short summary
==================
This test method tests ``assert.integer.unsigned.x.valueIsOdd``
of CNM_AssertionInterfaces library, 
it provides the possibility to handover test data via parameter 


.. <legal notes>

legal notes
=================
| SPDX-FileCopyrightText: © 2022 ekvip automation GmbH <info@ekvip.de>
| SPDX-License-Identifier: Apache-2.0
| For details check: Apache-2.0_

.. _Apache-2.0: https://www.apache.org/licenses/LICENSE-2.0

.. </legal notes>

parameters
==========

*)

METHOD testValueIsOdd
VAR_INPUT
	(* for the test it's the parameter ``currentValue`` *)
	valueToTest	:__UXINT;
END_VAR
VAR
	(* just the expectation if the assertion to test must be worng or true *)
	assertionIsWrong		:BOOL;
	(* contains the format string for the test message *)
	message					:Tc2_System.T_MaxString;
	(* TwinCAT printf with the test message *)
	messageStringBuilder	:Tc2_Utilities.FB_FormatString;
END_VAR
THIS^.assertorContainer.resetAssertor();

assertionIsWrong := (NOT valueToTest.FIRST_BIT);

message := SEL(
	assertionIsWrong,
	'currentValue is %d assertion must be TRUE',
	'currentValue is %d assertion must be FALSE'
);

messageStringBuilder(
	sFormat := message,
	arg1 := THIS^.AnyToArg(valueToTest)
);

THIS^.assertorContainer.assertor.assert.integer.unsigned.x.valueIsOdd(
	currentValue 	:= valueToTest,
	message			:= ''  
); 

THIS^.AssertEquals_BOOL(
	Expected 	:= assertionIsWrong,
	Actual 		:= THIS^.assertorContainer.wasAssertionWrong,
	Message 	:= messageStringBuilder.sOut
);
END_METHOD

END_FUNCTION_BLOCK

// ---- AssertionTester/AssertionTests/IntegerAssertions/classes/XintAssertionTests.TcPOU
(*

short summary
==================
This class tests all methods of xint assertions
with various combinations of inputs and checks expected 
outputs are satisfied or not

.. <legal notes>

legal notes
=================
| SPDX-FileCopyrightText: © 2022 ekvip automation GmbH <info@ekvip.de>
| SPDX-License-Identifier: Apache-2.0
| For details check: Apache-2.0_

.. _Apache-2.0: https://www.apache.org/licenses/LICENSE-2.0

.. </legal notes>

methods and properties
======================

*)

FUNCTION_BLOCK XintAssertionTests EXTENDS AbstractAssertorTest
VAR_INPUT
END_VAR
VAR CONSTANT
	(* prefix to unify the test names *)
	TEST_NAME_PREFIX	:Tc2_System.T_MaxString := 'assert.integer.signed.x.';
	(* number of the lsb *)
	FIRST_BIT				:USINT := 0;
	(* number of the msb *)
	LAST_BIT				:USINT := ((SIZEOF(__XINT)*8)-1);
	(* since we don't know the lenght of __XINT we need it to initialize ``MULTIPLICAND`` *)
	{attribute 'hide'}
	INIT_VALUE_MULTIPLICAND	:__XWORD := 16#1111_1111;
	(* multiplicand for the ``multiplier`` *)
	{warning disable C0196}
	MULTIPLICAND			:__XINT := (ROR(INIT_VALUE_MULTIPLICAND, 32) OR INIT_VALUE_MULTIPLICAND);
	{warning enable C0196}
	(* first of all multipliers the test iterates *)
	FIRST_MULTIPLIER		:__XINT := 0;
	(* first of all multipliers the test iterates *)
	LAST_MULTIPLIER			:__XINT := 15;
	(* just the value zero *)
	ZERO					:__XINT := 0;
	(* just the lsb is set, it's just the value one *)
	LSB_ONLY				:__XINT := 1;
	(* all bits are set *)
	ALL_BITS_SET			:__XINT := -1;
	(* the msb is set only *)
	MINIMUM_VALUE			:__XINT := ROR(LSB_ONLY,1);
	(* 
	since we don't know the lenght of __XINT 
	we need it to initialize ``MAXIMUM_VALUE``.
	SHR is not working with __XINT
	*)
	{attribute 'hide'}
	{warning disable C0195}
	BINARY_MINUS_ONE		:__XWORD := ALL_BITS_SET;
	{warning enable C0195}
	(* the msb is unset only *)
	{warning disable C0196}
	MAXIMUM_VALUE			:__XINT := SHR(BINARY_MINUS_ONE,1);
	{warning ensable C0196}
END_VAR

THIS^.runValueIsEqualToTests();
THIS^.runValueIsEvenTests();
THIS^.runValueIsGreaterTests();
THIS^.runValueIsInRangeOfTests();
THIS^.runValueIsLessThanTests();
THIS^.runValueIsMaxTests();
THIS^.runValueIsMinTests();
THIS^.runValueIsNegativeTests();
THIS^.runValueIsNotEqualToTests();
THIS^.runValueIsOddTests();
THIS^.runValueIsPositiveTests();

(*

short summary
==================
This test method is a helper function to create a unified test name

.. <legal notes>

legal notes
=================
| SPDX-FileCopyrightText: © 2022 ekvip automation GmbH <info@ekvip.de>
| SPDX-License-Identifier: Apache-2.0
| For details check: Apache-2.0_

.. _Apache-2.0: https://www.apache.org/licenses/LICENSE-2.0

.. </legal notes>

parameters
==========

*)

METHOD PROTECTED getTestNameFor :Tc2_System.T_MaxString
VAR_INPUT
	(* name of the method to test, to create a unified test name *)
	nameOfMethodToTest	:Tc2_System.T_MaxString;
END_VAR
getTestNameFor := Tc2_Standard.CONCAT(THIS^.TEST_NAME_PREFIX, nameOfMethodToTest);
END_METHOD

(*

short summary
==================
This test method tests ``assert.integer.signed.x.valueIsEqualTo``
method of CNM_AssertionInterfaces library with various inputs

.. <legal notes>

legal notes
=================
| SPDX-FileCopyrightText: © 2022 ekvip automation GmbH <info@ekvip.de>
| SPDX-License-Identifier: Apache-2.0
| For details check: Apache-2.0_

.. _Apache-2.0: https://www.apache.org/licenses/LICENSE-2.0

.. </legal notes>

*)

METHOD runValueIsEqualToTests
RETURN (NOT TcUnit.TEST_ORDERED(THIS^.getTestNameFor('valueIsEqualTo')));

THIS^.testValueIsEqualTo(
	valueToTest := THIS^.ZERO,
	expected := THIS^.ALL_BITS_SET
);
THIS^.testValueIsEqualTo(
	valueToTest := THIS^.ZERO,
	expected := THIS^.ZERO
);
THIS^.testValueIsEqualTo(
	valueToTest := THIS^.ALL_BITS_SET,
	expected := THIS^.ALL_BITS_SET
);
THIS^.testValueIsEqualTo(
	valueToTest := THIS^.ALL_BITS_SET,
	expected := THIS^.ZERO
);
THIS^.testValueIsEqualTo(
	valueToTest := THIS^.LSB_ONLY,
	expected := THIS^.LSB_ONLY
);
THIS^.testValueIsEqualTo(
	valueToTest := THIS^.LSB_ONLY,
	expected := THIS^.MINIMUM_VALUE
);
THIS^.testValueIsEqualTo(
	valueToTest := THIS^.MINIMUM_VALUE,
	expected := THIS^.MINIMUM_VALUE
);
THIS^.testValueIsEqualTo(
	valueToTest := THIS^.MINIMUM_VALUE,
	expected := THIS^.LSB_ONLY
);
THIS^.testValueIsEqualTo(
	valueToTest := THIS^.MINIMUM_VALUE,
	expected := THIS^.MAXIMUM_VALUE
);

TcUnit.TEST_FINISHED();
END_METHOD

(*

short summary
==================
This test method tests ``assert.integer.signed.x.valueIsEven``
of CNM_AssertionInterfaces library with various inputs

.. <legal notes>

legal notes
=================
| SPDX-FileCopyrightText: © 2022 ekvip automation GmbH <info@ekvip.de>
| SPDX-License-Identifier: Apache-2.0
| For details check: Apache-2.0_

.. _Apache-2.0: https://www.apache.org/licenses/LICENSE-2.0

.. </legal notes>

*)

METHOD runValueIsEvenTests
VAR
	(* it's just part of the test data *)
	valueToTest	:__XINT;
	(* multiplier to get various bit patterns *)
	multiplier	:__XINT;
END_VAR
RETURN (NOT TcUnit.TEST_ORDERED(THIS^.getTestNameFor('valueIsEven')));

FOR multiplier := THIS^.FIRST_MULTIPLIER TO THIS^.LAST_MULTIPLIER DO
	valueToTest := (THIS^.MULTIPLICAND * multiplier);
	THIS^.testValueIsEven(
		valueToTest := valueToTest
	);
END_FOR

TcUnit.TEST_FINISHED();
END_METHOD

(*

short summary
==================
This test method tests ``assert.integer.signed.x.valueIsGreaterThan``
method of CNM_AssertionInterfaces library with various inputs

.. <legal notes>

legal notes
=================
| SPDX-FileCopyrightText: © 2022 ekvip automation GmbH <info@ekvip.de>
| SPDX-License-Identifier: Apache-2.0
| For details check: Apache-2.0_

.. _Apache-2.0: https://www.apache.org/licenses/LICENSE-2.0

.. </legal notes>

*)

METHOD runValueIsGreaterTests
RETURN (NOT TcUnit.TEST_ORDERED(THIS^.getTestNameFor('valueIsGreaterThan')));

THIS^.testValueIsGreater(
	valueToTest := THIS^.ZERO,
	less := THIS^.ALL_BITS_SET
);
THIS^.testValueIsGreater(
	valueToTest := THIS^.ZERO,
	less := THIS^.ZERO
);
THIS^.testValueIsGreater(
	valueToTest := THIS^.ALL_BITS_SET,
	less := THIS^.ALL_BITS_SET
);
THIS^.testValueIsGreater(
	valueToTest := THIS^.ALL_BITS_SET,
	less := THIS^.ZERO
);
THIS^.testValueIsGreater(
	valueToTest := THIS^.LSB_ONLY,
	less := THIS^.LSB_ONLY
);
THIS^.testValueIsGreater(
	valueToTest := THIS^.LSB_ONLY,
	less := THIS^.ZERO
);
THIS^.testValueIsGreater(
	valueToTest := THIS^.LSB_ONLY,
	less := (THIS^.LSB_ONLY+THIS^.LSB_ONLY)
);
THIS^.testValueIsGreater(
	valueToTest := THIS^.MINIMUM_VALUE,
	less := THIS^.MINIMUM_VALUE
);
THIS^.testValueIsGreater(
	valueToTest := THIS^.MINIMUM_VALUE,
	less := THIS^.ALL_BITS_SET
);
THIS^.testValueIsGreater(
	valueToTest := THIS^.MINIMUM_VALUE,
	less := THIS^.MAXIMUM_VALUE
);
THIS^.testValueIsGreater(
	valueToTest := THIS^.MAXIMUM_VALUE,
	less := THIS^.MINIMUM_VALUE
);

TcUnit.TEST_FINISHED();
END_METHOD

(*

short summary
==================
This test method tests ``assert.integer.signed.x.valueIsInRangeOf``
method of CNM_AssertionInterfaces library with various inputs

.. <legal notes>

legal notes
=================
| SPDX-FileCopyrightText: © 2022 ekvip automation GmbH <info@ekvip.de>
| SPDX-License-Identifier: Apache-2.0
| For details check: Apache-2.0_

.. _Apache-2.0: https://www.apache.org/licenses/LICENSE-2.0

.. </legal notes>

*)

METHOD runValueIsInRangeOfTests
RETURN (NOT TcUnit.TEST_ORDERED(THIS^.getTestNameFor('valueIsInRangeOf')));

THIS^.testValueIsInRangeOf(
	lower := THIS^.ZERO,
	valueToTest := THIS^.LSB_ONLY,
	upper := THIS^.ALL_BITS_SET
);
THIS^.testValueIsInRangeOf(
	lower := THIS^.ZERO,
	valueToTest := THIS^.ZERO,
	upper := THIS^.ZERO
);
THIS^.testValueIsInRangeOf(
	lower := THIS^.ALL_BITS_SET,
	valueToTest := THIS^.ALL_BITS_SET,
	upper := THIS^.ALL_BITS_SET
);
THIS^.testValueIsInRangeOf(
	lower := THIS^.ALL_BITS_SET,
	valueToTest := THIS^.LSB_ONLY,
	upper := THIS^.ZERO
);
THIS^.testValueIsInRangeOf(
	lower := THIS^.ALL_BITS_SET,
	valueToTest := THIS^.ZERO,
	upper := THIS^.ZERO
);
THIS^.testValueIsInRangeOf(
	lower := THIS^.MAXIMUM_VALUE,
	valueToTest := THIS^.ZERO,
	upper := THIS^.MINIMUM_VALUE
);
THIS^.testValueIsInRangeOf(
	lower := THIS^.MINIMUM_VALUE,
	valueToTest := THIS^.ZERO,
	upper := THIS^.MAXIMUM_VALUE
);
THIS^.testValueIsInRangeOf(
	lower := THIS^.MAXIMUM_VALUE,
	valueToTest := THIS^.MINIMUM_VALUE,
	upper := THIS^.MINIMUM_VALUE
);
THIS^.testValueIsInRangeOf(
	lower := THIS^.MINIMUM_VALUE,
	valueToTest := THIS^.MAXIMUM_VALUE,
	upper := THIS^.MAXIMUM_VALUE
);
THIS^.testValueIsInRangeOf(
	lower := THIS^.MINIMUM_VALUE,
	valueToTest := THIS^.MINIMUM_VALUE,
	upper := THIS^.MAXIMUM_VALUE
);

TEST_FINISHED();
END_METHOD

(*

short summary
==================
This test method tests ``assert.integer.signed.x.valueIsLessThan``
method of CNM_AssertionInterfaces library with various inputs

.. <legal notes>

legal notes
=================
| SPDX-FileCopyrightText: © 2022 ekvip automation GmbH <info@ekvip.de>
| SPDX-License-Identifier: Apache-2.0
| For details check: Apache-2.0_

.. _Apache-2.0: https://www.apache.org/licenses/LICENSE-2.0

.. </legal notes>

*)

METHOD runValueIsLessThanTests
RETURN (NOT TcUnit.TEST_ORDERED(THIS^.getTestNameFor('valueIsLessThan')));

THIS^.testValueIsLessThan(
	valueToTest := THIS^.ZERO,
	greater := THIS^.ALL_BITS_SET
);
THIS^.testValueIsLessThan(
	valueToTest := THIS^.ZERO,
	greater := THIS^.ZERO
);
THIS^.testValueIsLessThan(
	valueToTest := THIS^.ALL_BITS_SET,
	greater := THIS^.ALL_BITS_SET
);
THIS^.testValueIsLessThan(
	valueToTest := THIS^.ALL_BITS_SET,
	greater := THIS^.ZERO
);
THIS^.testValueIsLessThan(
	valueToTest := THIS^.LSB_ONLY,
	greater := THIS^.LSB_ONLY
);
THIS^.testValueIsLessThan(
	valueToTest := THIS^.LSB_ONLY,
	greater := THIS^.ZERO
);
THIS^.testValueIsLessThan(
	valueToTest := THIS^.MINIMUM_VALUE,
	greater := (THIS^.MINIMUM_VALUE+THIS^.LSB_ONLY)
);
THIS^.testValueIsLessThan(
	valueToTest := THIS^.MINIMUM_VALUE,
	greater := THIS^.MINIMUM_VALUE
);
THIS^.testValueIsLessThan(
	valueToTest := THIS^.MINIMUM_VALUE,
	greater := THIS^.ALL_BITS_SET
);
THIS^.testValueIsLessThan(
	valueToTest := THIS^.MINIMUM_VALUE,
	greater := THIS^.MAXIMUM_VALUE
);
THIS^.testValueIsLessThan(
	valueToTest := THIS^.MAXIMUM_VALUE,
	greater := THIS^.MINIMUM_VALUE
);

TcUnit.TEST_FINISHED();
END_METHOD

(*

short summary
==================
This test method tests ``assert.integer.signed.x.valueIsMax``
method of CNM_AssertionInterfaces library with various inputs

.. <legal notes>

legal notes
=================
| SPDX-FileCopyrightText: © 2022 ekvip automation GmbH <info@ekvip.de>
| SPDX-License-Identifier: Apache-2.0
| For details check: Apache-2.0_

.. _Apache-2.0: https://www.apache.org/licenses/LICENSE-2.0

.. </legal notes>

*)

METHOD runValueIsMaxTests
RETURN (NOT TcUnit.TEST_ORDERED(THIS^.getTestNameFor('valueIsMax')));

THIS^.testValueIsMax(
	valueToTest := THIS^.ZERO,
	maximum := THIS^.LSB_ONLY
);
THIS^.testValueIsMax(
	valueToTest := THIS^.LSB_ONLY,
	maximum := THIS^.ZERO
);
THIS^.testValueIsMax(
	valueToTest := THIS^.ZERO,
	maximum := THIS^.ZERO
);
THIS^.testValueIsMax(
	valueToTest := THIS^.ALL_BITS_SET,
	maximum := ALL_BITS_SET
);
THIS^.testValueIsMax(
	valueToTest := (THIS^.ALL_BITS_SET-THIS^.LSB_ONLY),
	maximum := THIS^.ALL_BITS_SET
);
THIS^.testValueIsMax(
	valueToTest := THIS^.ALL_BITS_SET,
	maximum := (THIS^.ALL_BITS_SET-THIS^.LSB_ONLY)
);
THIS^.testValueIsMax(
	valueToTest := THIS^.MINIMUM_VALUE,
	maximum := (THIS^.MINIMUM_VALUE+THIS^.LSB_ONLY)
);
THIS^.testValueIsMax(
	valueToTest := (THIS^.MINIMUM_VALUE+THIS^.LSB_ONLY),
	maximum := THIS^.MINIMUM_VALUE
);
THIS^.testValueIsMax(
	valueToTest := THIS^.MINIMUM_VALUE,
	maximum := THIS^.MINIMUM_VALUE
);
THIS^.testValueIsMax(
	valueToTest := THIS^.MINIMUM_VALUE,
	maximum := THIS^.MAXIMUM_VALUE
);
THIS^.testValueIsMax(
	valueToTest := THIS^.MAXIMUM_VALUE,
	maximum := THIS^.MINIMUM_VALUE
);

TcUnit.TEST_FINISHED();
END_METHOD

(*

short summary
==================
This test method tests ``assert.integer.signed.x.valueIsMin``
method of CNM_AssertionInterfaces library with various inputs

.. <legal notes>

legal notes
=================
| SPDX-FileCopyrightText: © 2022 ekvip automation GmbH <info@ekvip.de>
| SPDX-License-Identifier: Apache-2.0
| For details check: Apache-2.0_

.. _Apache-2.0: https://www.apache.org/licenses/LICENSE-2.0

.. </legal notes>

*)

METHOD runValueIsMinTests
RETURN (NOT TcUnit.TEST_ORDERED(THIS^.getTestNameFor('valueIsMin')));

THIS^.testValueIsMin(
	valueToTest := THIS^.ZERO,
	minimum := THIS^.LSB_ONLY
);
THIS^.testValueIsMin(
	valueToTest := THIS^.LSB_ONLY,
	minimum := THIS^.ZERO
);
THIS^.testValueIsMin(
	valueToTest := THIS^.ZERO,
	minimum := THIS^.ZERO
);
THIS^.testValueIsMin(
	valueToTest := THIS^.ALL_BITS_SET,
	minimum := ALL_BITS_SET
);
THIS^.testValueIsMin(
	valueToTest := (THIS^.ALL_BITS_SET-THIS^.LSB_ONLY),
	minimum := THIS^.ALL_BITS_SET
);
THIS^.testValueIsMin(
	valueToTest := THIS^.ALL_BITS_SET,
	minimum := (THIS^.ALL_BITS_SET-THIS^.LSB_ONLY)
);
THIS^.testValueIsMin(
	valueToTest := THIS^.MINIMUM_VALUE,
	minimum := (THIS^.MINIMUM_VALUE+THIS^.LSB_ONLY)
);
THIS^.testValueIsMin(
	valueToTest := (THIS^.MINIMUM_VALUE+THIS^.LSB_ONLY),
	minimum := THIS^.MINIMUM_VALUE
);
THIS^.testValueIsMin(
	valueToTest := THIS^.MINIMUM_VALUE,
	minimum := THIS^.MINIMUM_VALUE
);
THIS^.testValueIsMin(
	valueToTest := THIS^.MINIMUM_VALUE,
	minimum := THIS^.MAXIMUM_VALUE
);
THIS^.testValueIsMin(
	valueToTest := THIS^.MAXIMUM_VALUE,
	minimum := THIS^.MINIMUM_VALUE
);

TcUnit.TEST_FINISHED();
END_METHOD

(*

short summary
==================
This test method tests ``assert.integer.signed.x.valueIsNegative``
of CNM_AssertionInterfaces library with various inputs

.. <legal notes>

legal notes
=================
| SPDX-FileCopyrightText: © 2022 ekvip automation GmbH <info@ekvip.de>
| SPDX-License-Identifier: Apache-2.0
| For details check: Apache-2.0_

.. _Apache-2.0: https://www.apache.org/licenses/LICENSE-2.0

.. </legal notes>

*)

METHOD runValueIsNegativeTests
VAR
	(* it's just part of the test data *)
	valueToTest	:__XINT;
	(* multiplier to get various bit patterns *)
	multiplier	:__XINT;
END_VAR
RETURN (NOT TcUnit.TEST_ORDERED(THIS^.getTestNameFor('valueIsNegative')));

FOR multiplier := THIS^.FIRST_MULTIPLIER TO THIS^.LAST_MULTIPLIER DO
	valueToTest := (THIS^.MULTIPLICAND * multiplier);
	THIS^.testValueIsNegative(
		valueToTest := valueToTest
	);
END_FOR

TcUnit.TEST_FINISHED();
END_METHOD

(*

short summary
==================
This test method tests ``assert.integer.signed.x.valueIsNotEqualTo``
method of CNM_AssertionInterfaces library with various inputs

.. <legal notes>

legal notes
=================
| SPDX-FileCopyrightText: © 2022 ekvip automation GmbH <info@ekvip.de>
| SPDX-License-Identifier: Apache-2.0
| For details check: Apache-2.0_

.. _Apache-2.0: https://www.apache.org/licenses/LICENSE-2.0

.. </legal notes>

*)

METHOD runValueIsNotEqualToTests
RETURN (NOT TcUnit.TEST_ORDERED(THIS^.getTestNameFor('valueIsNotEqualTo')));

THIS^.testValueIsNotEqualTo(
	valueToTest := THIS^.ZERO,
	unexpected := THIS^.ALL_BITS_SET
);
THIS^.testValueIsNotEqualTo(
	valueToTest := THIS^.ZERO,
	unexpected := THIS^.ZERO
);
THIS^.testValueIsNotEqualTo(
	valueToTest := THIS^.ALL_BITS_SET,
	unexpected := THIS^.ALL_BITS_SET
);
THIS^.testValueIsNotEqualTo(
	valueToTest := THIS^.ALL_BITS_SET,
	unexpected := THIS^.ZERO
);
THIS^.testValueIsNotEqualTo(
	valueToTest := THIS^.LSB_ONLY,
	unexpected := THIS^.LSB_ONLY
);
THIS^.testValueIsNotEqualTo(
	valueToTest := THIS^.LSB_ONLY,
	unexpected := THIS^.MINIMUM_VALUE
);
THIS^.testValueIsNotEqualTo(
	valueToTest := THIS^.MINIMUM_VALUE,
	unexpected := THIS^.MINIMUM_VALUE
);
THIS^.testValueIsNotEqualTo(
	valueToTest := THIS^.MINIMUM_VALUE,
	unexpected := THIS^.LSB_ONLY
);
THIS^.testValueIsNotEqualTo(
	valueToTest := THIS^.MINIMUM_VALUE,
	unexpected := THIS^.MAXIMUM_VALUE
);

TcUnit.TEST_FINISHED();
END_METHOD

(*

short summary
==================
This test method tests ``assert.integer.signed.x.valueIsOdd``
of CNM_AssertionInterfaces library with various inputs

.. <legal notes>

legal notes
=================
| SPDX-FileCopyrightText: © 2022 ekvip automation GmbH <info@ekvip.de>
| SPDX-License-Identifier: Apache-2.0
| For details check: Apache-2.0_

.. _Apache-2.0: https://www.apache.org/licenses/LICENSE-2.0

.. </legal notes>

*)

METHOD runValueIsOddTests
VAR
	(* it's just part of the test data *)
	valueToTest	:__XINT;
	(* multiplier to get various bit patterns *)
	multiplier	:__XINT;
END_VAR
RETURN (NOT TcUnit.TEST_ORDERED(THIS^.getTestNameFor('valueIsOdd')));

FOR multiplier := THIS^.FIRST_MULTIPLIER TO THIS^.LAST_MULTIPLIER DO
	valueToTest := (THIS^.MULTIPLICAND * multiplier);
	THIS^.testValueIsOdd(
		valueToTest := valueToTest
	);
END_FOR

TcUnit.TEST_FINISHED();
END_METHOD

(*

short summary
==================
This test method tests ``assert.integer.signed.x.valueIsPositive``
of CNM_AssertionInterfaces library with various inputs

.. <legal notes>

legal notes
=================
| SPDX-FileCopyrightText: © 2022 ekvip automation GmbH <info@ekvip.de>
| SPDX-License-Identifier: Apache-2.0
| For details check: Apache-2.0_

.. _Apache-2.0: https://www.apache.org/licenses/LICENSE-2.0

.. </legal notes>

*)

METHOD runValueIsPositiveTests
VAR
	(* it's just part of the test data *)
	valueToTest	:__XINT;
	(* multiplier to get various bit patterns *)
	multiplier	:__XINT;
END_VAR
RETURN (NOT TcUnit.TEST_ORDERED(THIS^.getTestNameFor('valueIsPositive')));

FOR multiplier := THIS^.FIRST_MULTIPLIER TO THIS^.LAST_MULTIPLIER DO
	valueToTest := (THIS^.MULTIPLICAND * multiplier);
	THIS^.testValueIsPositive(
		valueToTest := valueToTest
	);
END_FOR

TcUnit.TEST_FINISHED();
END_METHOD

(*

short summary
==================
This test method tests ``assert.integer.signed.x.valueIsEqualTo``
method of CNM_AssertionInterfaces library, 
it provides the possibility to handover test data via parameter 


.. <legal notes>

legal notes
=================
| SPDX-FileCopyrightText: © 2022 ekvip automation GmbH <info@ekvip.de>
| SPDX-License-Identifier: Apache-2.0
| For details check: Apache-2.0_

.. _Apache-2.0: https://www.apache.org/licenses/LICENSE-2.0

.. </legal notes>

parameters
==========

*)

METHOD testValueIsEqualTo
VAR_INPUT
	(* for the test it's the parameter ``currentValue`` *)
	valueToTest	:__XINT;
	(* for the test it's the parameter ``expectedValue`` *)
	expected	:__XINT;
END_VAR
VAR
	(* just the expectation if the assertion to test must be worng or true *)
	assertionIsWrong		:BOOL;
	(* contains the format string for the test message *)
	message					:Tc2_System.T_MaxString;
	(* TwinCAT printf with the test message *)
	messageStringBuilder	:Tc2_Utilities.FB_FormatString;
END_VAR
THIS^.assertorContainer.resetAssertor();

assertionIsWrong := (valueToTest <> expected);
message := SEL(
	assertionIsWrong,
	'currentValue is %d expectedValue is %d assertion must be TRUE', 
	'currentValue is %d expectedValue is %d assertion must be FALSE'
);
messageStringBuilder(
	sFormat := message,
	arg1 := THIS^.AnyToArg(valueToTest),
	arg2 := THIS^.AnyToArg(expected)
);

THIS^.assertorContainer.assertor.assert.integer.signed.x.valueIsEqualTo(
	currentValue := valueToTest,
	expectedValue := expected,
	message := ''
);

THIS^.AssertEquals_BOOL(
	Expected 	:= assertionIsWrong,
	Actual 		:= THIS^.assertorContainer.wasAssertionWrong,
	Message 	:= messageStringBuilder.sOut
);
END_METHOD

(*

short summary
==================
This test method tests ``assert.integer.signed.x.valueIsEven``
of CNM_AssertionInterfaces library, 
it provides the possibility to handover test data via parameter 


.. <legal notes>

legal notes
=================
| SPDX-FileCopyrightText: © 2022 ekvip automation GmbH <info@ekvip.de>
| SPDX-License-Identifier: Apache-2.0
| For details check: Apache-2.0_

.. _Apache-2.0: https://www.apache.org/licenses/LICENSE-2.0

.. </legal notes>

parameters
==========

*)

METHOD testValueIsEven
VAR_INPUT
	(* for the test it's the parameter ``currentValue`` *)
	valueToTest	:__XINT;
END_VAR
VAR
	(* just the expectation if the assertion to test must be worng or true *)
	assertionIsWrong		:BOOL;
	(* contains the format string for the test message *)
	message					:Tc2_System.T_MaxString;
	(* TwinCAT printf with the test message *)
	messageStringBuilder	:Tc2_Utilities.FB_FormatString;
END_VAR
THIS^.assertorContainer.resetAssertor();

assertionIsWrong := (valueToTest.FIRST_BIT);

message := SEL(
	assertionIsWrong,
	'currentValue is %d assertion must be TRUE',
	'currentValue is %d assertion must be FALSE'
);

messageStringBuilder(
	sFormat := message,
	arg1 := THIS^.AnyToArg(valueToTest)
);

THIS^.assertorContainer.assertor.assert.integer.signed.x.valueIsEven(
	currentValue 	:= valueToTest,
	message			:= ''  
); 

THIS^.AssertEquals_BOOL(
	Expected 	:= assertionIsWrong,
	Actual 		:= THIS^.assertorContainer.wasAssertionWrong,
	Message 	:= messageStringBuilder.sOut
);
END_METHOD

(*

short summary
==================
This test method tests ``assert.integer.signed.x.valueIsGreaterThan``
method of CNM_AssertionInterfaces library, 
it provides the possibility to handover test data via parameter 


.. <legal notes>

legal notes
=================
| SPDX-FileCopyrightText: © 2022 ekvip automation GmbH <info@ekvip.de>
| SPDX-License-Identifier: Apache-2.0
| For details check: Apache-2.0_

.. _Apache-2.0: https://www.apache.org/licenses/LICENSE-2.0

.. </legal notes>

parameters
==========

*)

METHOD testValueIsGreater
VAR_INPUT
	(* for the test it's the parameter ``currentValue`` *)
	valueToTest	:__XINT;
	(* for the test it's the parameter ``lessValue`` *)
	less		:__XINT;
END_VAR
VAR
	(* just the expectation if the assertion to test must be worng or true *)
	assertionIsWrong		:BOOL;
	(* contains the format string for the test message *)
	message					:Tc2_System.T_MaxString;
	(* TwinCAT printf with the test message *)
	messageStringBuilder	:Tc2_Utilities.FB_FormatString;
END_VAR
THIS^.assertorContainer.resetAssertor();

assertionIsWrong := (valueToTest <= less);
message := SEL(
	assertionIsWrong,
	'currentValue is %d lessValue is %d assertion must be TRUE', 
	'currentValue is %d lessValue is %d assertion must be FALSE'
);
messageStringBuilder(
	sFormat := message,
	arg1 := THIS^.AnyToArg(valueToTest),
	arg2 := THIS^.AnyToArg(less)
);

THIS^.assertorContainer.assertor.assert.integer.signed.x.valueIsGreaterThan(
	currentValue := valueToTest,
	lessValue := less,
	message := ''
);

THIS^.AssertEquals_BOOL(
	Expected 	:= assertionIsWrong,
	Actual 		:= THIS^.assertorContainer.wasAssertionWrong,
	Message 	:= messageStringBuilder.sOut
);
END_METHOD

(*

short summary
==================
This test method tests ``assert.integer.signed.x.valueIsInRangeOf``
method of CNM_AssertionInterfaces library, 
it provides the possibility to handover test data via parameter 


.. <legal notes>

legal notes
=================
| SPDX-FileCopyrightText: © 2022 ekvip automation GmbH <info@ekvip.de>
| SPDX-License-Identifier: Apache-2.0
| For details check: Apache-2.0_

.. _Apache-2.0: https://www.apache.org/licenses/LICENSE-2.0

.. </legal notes>

parameters
==========

*)

METHOD testValueIsInRangeOf
VAR_INPUT
	(* for the test it's the parameter ``lowerLimit`` *)
	lower		:__XINT;
	(* for the test it's the parameter ``currentValue`` *)
	valueToTest	:__XINT;
	(* for the test it's the parameter ``upperLimit`` *)
	upper		:__XINT;
END_VAR          
VAR
	(* just the expectation if the assertion to test must be worng or true *)
	assertionIsWrong		:BOOL;
	(* contains the format string for the test message *)
	message					:Tc2_System.T_MaxString;
	(* TwinCAT printf with the test message *)
	messageStringBuilder	:Tc2_Utilities.FB_FormatString;
END_VAR
THIS^.assertorContainer.resetAssertor();

assertionIsWrong := ((valueToTest < lower) OR (valueToTest > upper)); 

message := SEL(
	assertionIsWrong,
	'lowerLimit is %d currentValue is %d upperLimit is %d assertion must be TRUE', 
	'lowerLimit is %d currentValue is %d upperLimit is %d assertion must be FALSE'
);

messageStringBuilder(
	sFormat := message,
	arg1 := THIS^.AnyToArg(lower),
	arg2 := THIS^.AnyToArg(valueToTest),
	arg3 := THIS^.AnyToArg(upper)
);

THIS^.assertorContainer.assertor.assert.integer.signed.x.valueIsInRangeOf(
	lowerLimit := lower,
	currentValue := valueToTest,
	upperLimit := upper,
	message := ''
);

THIS^.AssertEquals_BOOL(
	Expected 	:= assertionIsWrong,
	Actual 		:= THIS^.assertorContainer.wasAssertionWrong,
	Message 	:= messageStringBuilder.sOut
);
END_METHOD

(*

short summary
==================
This test method tests ``assert.integer.signed.x.valueIsLessThan``
method of CNM_AssertionInterfaces library, 
it provides the possibility to handover test data via parameter 


.. <legal notes>

legal notes
=================
| SPDX-FileCopyrightText: © 2022 ekvip automation GmbH <info@ekvip.de>
| SPDX-License-Identifier: Apache-2.0
| For details check: Apache-2.0_

.. _Apache-2.0: https://www.apache.org/licenses/LICENSE-2.0

.. </legal notes>

parameters
==========

*)

METHOD testValueIsLessThan
VAR_INPUT
	(* for the test it's the parameter ``currentValue`` *)
	valueToTest	:__XINT;
	(* for the test it's the parameter ``greaterValue`` *)
	greater		:__XINT;
END_VAR
VAR
	(* just the expectation if the assertion to test must be worng or true *)
	assertionIsWrong		:BOOL;
	(* contains the format string for the test message *)
	message					:Tc2_System.T_MaxString;
	(* TwinCAT printf with the test message *)
	messageStringBuilder	:Tc2_Utilities.FB_FormatString;
END_VAR
THIS^.assertorContainer.resetAssertor();

assertionIsWrong := (valueToTest >= greater);
message := SEL(
	assertionIsWrong,
	'currentValue is %d greaterValue is %d assertion must be TRUE',
	'currentValue is %d greaterValue is %d assertion must be FALSE'
);
messageStringBuilder(
	sFormat := message,
	arg1 := THIS^.AnyToArg(valueToTest),
	arg2 := THIS^.AnyToArg(greater)
);

THIS^.assertorContainer.assertor.assert.integer.signed.x.valueIsLessThan(
	currentValue := valueToTest,
	greaterValue := greater,
	message := ''
);

THIS^.AssertEquals_BOOL(
	Expected 	:= assertionIsWrong,
	Actual 		:= THIS^.assertorContainer.wasAssertionWrong,
	Message 	:= messageStringBuilder.sOut
);
END_METHOD

(*

short summary
==================
This test method tests ``assert.integer.signed.x.valueIsMax``
method of CNM_AssertionInterfaces library, 
it provides the possibility to handover test data via parameter 


.. <legal notes>

legal notes
=================
| SPDX-FileCopyrightText: © 2022 ekvip automation GmbH <info@ekvip.de>
| SPDX-License-Identifier: Apache-2.0
| For details check: Apache-2.0_

.. _Apache-2.0: https://www.apache.org/licenses/LICENSE-2.0

.. </legal notes>

parameters
==========

*)

METHOD testValueIsMax 
VAR_INPUT
	(* for the test it's the parameter ``currentValue`` *)
	valueToTest	:__XINT;
	(* for the test it's the parameter ``maximumValue`` *)
	maximum		:__XINT;
END_VAR
VAR
	(* just the expectation if the assertion to test must be worng or true *)
	assertionIsWrong		:BOOL;
	(* contains the format string for the test message *)
	message					:Tc2_System.T_MaxString;
	(* TwinCAT printf with the test message *)
	messageStringBuilder	:Tc2_Utilities.FB_FormatString;
END_VAR
THIS^.assertorContainer.resetAssertor();

assertionIsWrong := (valueToTest > maximum);
message := SEL(
	assertionIsWrong,
	'currentValue is %d maximumValue is %d assertion must be TRUE',
	'currentValue is %d maximumValue is %d assertion must be FALSE'
);
messageStringBuilder(
	sFormat := message,
	arg1 := THIS^.AnyToArg(valueToTest),
	arg2 := THIS^.AnyToArg(maximum)
);

THIS^.assertorContainer.assertor.assert.integer.signed.x.valueIsMax(
	currentValue := valueToTest,
	maximumValue := maximum,
	message := ''
);

THIS^.AssertEquals_BOOL(
	Expected 	:= assertionIsWrong,
	Actual 		:= THIS^.assertorContainer.wasAssertionWrong,
	Message 	:= messageStringBuilder.sOut
);
END_METHOD

(*

short summary
==================
This test method tests ``assert.integer.signed.x.valueIsMin``
method of CNM_AssertionInterfaces library, 
it provides the possibility to handover test data via parameter 


.. <legal notes>

legal notes
=================
| SPDX-FileCopyrightText: © 2022 ekvip automation GmbH <info@ekvip.de>
| SPDX-License-Identifier: Apache-2.0
| For details check: Apache-2.0_

.. _Apache-2.0: https://www.apache.org/licenses/LICENSE-2.0

.. </legal notes>

parameters
==========

*)

METHOD testValueIsMin 
VAR_INPUT
	(* for the test it's the parameter ``currentValue`` *)
	valueToTest	:__XINT;
	(* for the test it's the parameter ``minimumValue`` *)
	minimum		:__XINT;
END_VAR
VAR
	(* just the expectation if the assertion to test must be worng or true *)
	assertionIsWrong		:BOOL;
	(* contains the format string for the test message *)
	message					:Tc2_System.T_MaxString;
	(* TwinCAT printf with the test message *)
	messageStringBuilder	:Tc2_Utilities.FB_FormatString;
END_VAR
THIS^.assertorContainer.resetAssertor();

assertionIsWrong := (valueToTest < minimum);
message := SEL(
	assertionIsWrong,
	'currentValue is %d minimumValue is %d assertion must be TRUE',
	'currentValue is %d minimumValue is %d assertion must be FALSE'
);
messageStringBuilder(
	sFormat := message,
	arg1 := THIS^.AnyToArg(valueToTest),
	arg2 := THIS^.AnyToArg(minimum)
);

THIS^.assertorContainer.assertor.assert.integer.signed.x.valueIsMin(
	currentValue := valueToTest,
	minimumValue := minimum,
	message := ''
);

THIS^.AssertEquals_BOOL(
	Expected 	:= assertionIsWrong,
	Actual 		:= THIS^.assertorContainer.wasAssertionWrong,
	Message 	:= messageStringBuilder.sOut
);
END_METHOD

(*

short summary
==================
This test method tests ``assert.integer.signed.x.valueIsNegative``
of CNM_AssertionInterfaces library, 
it provides the possibility to handover test data via parameter 


.. <legal notes>

legal notes
=================
| SPDX-FileCopyrightText: © 2022 ekvip automation GmbH <info@ekvip.de>
| SPDX-License-Identifier: Apache-2.0
| For details check: Apache-2.0_

.. _Apache-2.0: https://www.apache.org/licenses/LICENSE-2.0

.. </legal notes>

parameters
==========

*)

METHOD testValueIsNegative
VAR_INPUT
	(* for the test it's the parameter ``currentValue`` *)
	valueToTest	:__XINT;
END_VAR
VAR
	(* just the expectation if the assertion to test must be worng or true *)
	assertionIsWrong		:BOOL;
	(* contains the format string for the test message *)
	message					:Tc2_System.T_MaxString;
	(* TwinCAT printf with the test message *)
	messageStringBuilder	:Tc2_Utilities.FB_FormatString;
END_VAR
THIS^.assertorContainer.resetAssertor();

assertionIsWrong := (valueToTest >= THIS^.ZERO);

message := SEL(
	assertionIsWrong,
	'currentValue is %d assertion must be TRUE',
	'currentValue is %d assertion must be FALSE'
);

messageStringBuilder(
	sFormat := message,
	arg1 := THIS^.AnyToArg(valueToTest)
);

THIS^.assertorContainer.assertor.assert.integer.signed.x.valueIsNegative(
	currentValue 	:= valueToTest,
	message			:= ''  
); 

THIS^.AssertEquals_BOOL(
	Expected 	:= assertionIsWrong,
	Actual 		:= THIS^.assertorContainer.wasAssertionWrong,
	Message 	:= messageStringBuilder.sOut
);
END_METHOD

(*

short summary
==================
This test method tests ``assert.integer.signed.x.valueIsNotEqualTo``
method of CNM_AssertionInterfaces library, 
it provides the possibility to handover test data via parameter 


.. <legal notes>

legal notes
=================
| SPDX-FileCopyrightText: © 2022 ekvip automation GmbH <info@ekvip.de>
| SPDX-License-Identifier: Apache-2.0
| For details check: Apache-2.0_

.. _Apache-2.0: https://www.apache.org/licenses/LICENSE-2.0

.. </legal notes>

parameters
==========

*)

METHOD testValueIsNotEqualTo
VAR_INPUT
	(* for the test it's the parameter ``currentValue`` *)
	valueToTest	:__XINT;
	(* for the test it's the parameter ``unexpectedValue`` *)
	unexpected	:__XINT;
END_VAR
VAR
	(* just the expectation if the assertion to test must be worng or true *)
	assertionIsWrong		:BOOL;
	(* contains the format string for the test message *)
	message					:Tc2_System.T_MaxString;
	(* TwinCAT printf with the test message *)
	messageStringBuilder	:Tc2_Utilities.FB_FormatString;
END_VAR
THIS^.assertorContainer.resetAssertor();

assertionIsWrong := (valueToTest = unexpected);
message := SEL(
	assertionIsWrong,
	'currentValue is %d unexpectedValue is %d assertion must be TRUE', 
	'currentValue is %d unexpectedValue is %d assertion must be FALSE'
);
messageStringBuilder(
	sFormat := message,
	arg1 := THIS^.AnyToArg(valueToTest),
	arg2 := THIS^.AnyToArg(unexpected)
);

THIS^.assertorContainer.assertor.assert.integer.signed.x.valueIsNotEqualTo(
	currentValue := valueToTest,
	unexpectedValue := unexpected,
	message := ''
);

THIS^.AssertEquals_BOOL(
	Expected 	:= assertionIsWrong,
	Actual 		:= THIS^.assertorContainer.wasAssertionWrong,
	Message 	:= messageStringBuilder.sOut
);
END_METHOD

(*

short summary
==================
This test method tests ``assert.integer.signed.x.valueIsOdd``
of CNM_AssertionInterfaces library, 
it provides the possibility to handover test data via parameter 


.. <legal notes>

legal notes
=================
| SPDX-FileCopyrightText: © 2022 ekvip automation GmbH <info@ekvip.de>
| SPDX-License-Identifier: Apache-2.0
| For details check: Apache-2.0_

.. _Apache-2.0: https://www.apache.org/licenses/LICENSE-2.0

.. </legal notes>

parameters
==========

*)

METHOD testValueIsOdd
VAR_INPUT
	(* for the test it's the parameter ``currentValue`` *)
	valueToTest	:__XINT;
END_VAR
VAR
	(* just the expectation if the assertion to test must be worng or true *)
	assertionIsWrong		:BOOL;
	(* contains the format string for the test message *)
	message					:Tc2_System.T_MaxString;
	(* TwinCAT printf with the test message *)
	messageStringBuilder	:Tc2_Utilities.FB_FormatString;
END_VAR
THIS^.assertorContainer.resetAssertor();

assertionIsWrong := (NOT valueToTest.FIRST_BIT);

message := SEL(
	assertionIsWrong,
	'currentValue is %d assertion must be TRUE',
	'currentValue is %d assertion must be FALSE'
);

messageStringBuilder(
	sFormat := message,
	arg1 := THIS^.AnyToArg(valueToTest)
);

THIS^.assertorContainer.assertor.assert.integer.signed.x.valueIsOdd(
	currentValue 	:= valueToTest,
	message			:= ''  
); 

THIS^.AssertEquals_BOOL(
	Expected 	:= assertionIsWrong,
	Actual 		:= THIS^.assertorContainer.wasAssertionWrong,
	Message 	:= messageStringBuilder.sOut
);
END_METHOD

(*

short summary
==================
This test method tests ``assert.integer.signed.x.valueIsPositive``
of CNM_AssertionInterfaces library, 
it provides the possibility to handover test data via parameter 


.. <legal notes>

legal notes
=================
| SPDX-FileCopyrightText: © 2022 ekvip automation GmbH <info@ekvip.de>
| SPDX-License-Identifier: Apache-2.0
| For details check: Apache-2.0_

.. _Apache-2.0: https://www.apache.org/licenses/LICENSE-2.0

.. </legal notes>

parameters
==========

*)

METHOD testValueIsPositive
VAR_INPUT
	(* for the test it's the parameter ``currentValue`` *)
	valueToTest	:__XINT;
END_VAR
VAR
	(* just the expectation if the assertion to test must be worng or true *)
	assertionIsWrong		:BOOL;
	(* contains the format string for the test message *)
	message					:Tc2_System.T_MaxString;
	(* TwinCAT printf with the test message *)
	messageStringBuilder	:Tc2_Utilities.FB_FormatString;
END_VAR
THIS^.assertorContainer.resetAssertor();

assertionIsWrong := (valueToTest < THIS^.ZERO);

message := SEL(
	assertionIsWrong,
	'currentValue is %d assertion must be TRUE',
	'currentValue is %d assertion must be FALSE'
);

messageStringBuilder(
	sFormat := message,
	arg1 := THIS^.AnyToArg(valueToTest)
);

THIS^.assertorContainer.assertor.assert.integer.signed.x.valueIsPositive(
	currentValue 	:= valueToTest,
	message			:= ''  
); 

THIS^.AssertEquals_BOOL(
	Expected 	:= assertionIsWrong,
	Actual 		:= THIS^.assertorContainer.wasAssertionWrong,
	Message 	:= messageStringBuilder.sOut
);
END_METHOD

END_FUNCTION_BLOCK

// ---- AssertionTester/AssertionTests/ObjectAssertions/classes/internal/ConcreteObject.TcPOU
(*

short summary
==================
Wraper Class for Object to make ´´isObjectValid()´´ calls possible
needed because ´´AbstractAssertorTest´´ already extends ´´FB_TestSuite´´

.. <legal notes>

legal notes
=================
| SPDX-FileCopyrightText: © 2022 ekvip automation GmbH <info@ekvip.de>
| SPDX-License-Identifier: Apache-2.0
| For details check: Apache-2.0_

.. _Apache-2.0: https://www.apache.org/licenses/LICENSE-2.0

.. </legal notes>

*)
FUNCTION_BLOCK ConcreteObject EXTENDS CNM_AbstractObject.Object
VAR
END_VAR

(*

short summary
=================
This abstract property returns the class name of the concrete object, 
which is useful to check the class name for ``__DELETE``.

.. <legal notes>

legal notes
=================
| SPDX-FileCopyrightText: © 2022 ekvip automation GmbH <info@ekvip.de>
| SPDX-License-Identifier: Apache-2.0
| For details check: Apache-2.0_

.. _Apache-2.0: https://www.apache.org/licenses/LICENSE-2.0

.. </legal notes>

*)


PROPERTY className : CNM_AbstractObject.ClassName
GET
className := 'ConcreteObject_Internal';
END_GET
END_PROPERTY

END_FUNCTION_BLOCK

// ---- AssertionTester/AssertionTests/ObjectAssertions/classes/internal/DWordValue.TcPOU
(*

short summary
==================
Implementaion of CNM_AbstractObject.IObject for testing purposes

.. <legal notes>

legal notes
=================
| SPDX-FileCopyrightText: © 2022 ekvip automation GmbH <info@ekvip.de>
| SPDX-License-Identifier: Apache-2.0
| For details check: Apache-2.0_

.. _Apache-2.0: https://www.apache.org/licenses/LICENSE-2.0

.. </legal notes>

*)

FUNCTION_BLOCK DWordValue EXTENDS CNM_AbstractObject.Object IMPLEMENTS IDWord

VAR
	(* local DWORD value of this Class*)
	dwordValue :DWORD;
END_VAR

(*

short summary
=================
This abstract property returns the class name of the concrete object, 
which is useful to check the class name for ``__DELETE``.

.. <legal notes>

legal notes
=================
| SPDX-FileCopyrightText: © 2022 ekvip automation GmbH <info@ekvip.de>
| SPDX-License-Identifier: Apache-2.0
| For details check: Apache-2.0_

.. _Apache-2.0: https://www.apache.org/licenses/LICENSE-2.0

.. </legal notes>

*)


PROPERTY className : CNM_AbstractObject.ClassName
GET
className := 'DWordValue_Internal';
END_GET
END_PROPERTY

(*

short summary
=================
overwrites compareTo of IObject: This method compares a foreign object with the own one, this is needed for sort orders.

.. <legal notes>

legal notes
=================
| SPDX-FileCopyrightText: © 2022 ekvip automation GmbH <info@ekvip.de>
| SPDX-License-Identifier: Apache-2.0
| For details check: Apache-2.0_

.. _Apache-2.0: https://www.apache.org/licenses/LICENSE-2.0

.. </legal notes>

parameters
=================
:return:``SMALLER``: ``THIS`` precedes in order,
``EQUAL``: ``THIS`` and ``object`` at the same position in order,
``GREATER``: ``THIS`` is after in order.
Checkout the library CNM_ReturnTypes.

*)

METHOD compareTo :CNM_ReturnTypes.ComparationResult
VAR_INPUT
	(* foreign objet to compare*)
	object		:CNM_AbstractObject.IObject;
END_VAR
VAR
	dwordObject	:IDWord;
END_VAR
IF (__QUERYINTERFACE(object, dwordObject)) THEN
	IF (THIS^.value < dwordObject.value) THEN
		compareTo := CNM_ReturnTypes.ComparationResult.SMALLER;
	ELSIF (THIS^.value = dwordObject.value) THEN
		compareTo := CNM_ReturnTypes.ComparationResult.EQUAL;
	ELSE
		compareTo := CNM_ReturnTypes.ComparationResult.GREATER;
	END_IF
ELSE
	compareTo := CNM_ReturnTypes.ComparationResult.SMALLER;
END_IF
END_METHOD

(*

short summary
=================
For initializing an DWordValue

.. <legal notes>

legal notes
=================
| SPDX-FileCopyrightText: © 2022 ekvip automation GmbH <info@ekvip.de>
| SPDX-License-Identifier: Apache-2.0
| For details check: Apache-2.0_

.. _Apache-2.0: https://www.apache.org/licenses/LICENSE-2.0

.. </legal notes>

parameters
=================

*)


METHOD FB_Init: BOOL
VAR_INPUT
	(* if TRUE, the retain variables are initialized (warm start / cold start) *)
    bInitRetains	:BOOL;
	(* if TRUE, the instance afterwards gets moved into the copy code (online change) *)
    bInCopyCode		:BOOL;
	(* value of the DWordValue Class*)
	initvalue 		:DWORD;
END_VAR
THIS^.dwordValue := initvalue;
END_METHOD

(*

short summary
=============
contains the DWORD Value of this Class

.. <legal notes>

legal notes
=================
| SPDX-FileCopyrightText: © 2023 ekvip automation GmbH <info@ekvip.de>
| SPDX-License-Identifier: Apache-2.0
| For details check: Apache-2.0_

.. _Apache-2.0: https://www.apache.org/licenses/LICENSE-2.0

.. </legal notes>

*)

PROPERTY value : DWORD
GET
value := THIS^.dwordValue;
END_GET
SET
THIS^.value := dwordValue;
END_SET
END_PROPERTY

END_FUNCTION_BLOCK

// ---- AssertionTester/AssertionTests/ObjectAssertions/classes/internal/ReverseOrderComparator.TcPOU
(*

short summary
=================
A comparator to reverse the natural order of the objects

.. <legal notes>

legal notes
=================
| SPDX-FileCopyrightText: © 2024 ekvip automation GmbH <info@ekvip.de>
| SPDX-License-Identifier: Apache-2.0
| For details check: Apache-2.0_

.. _Apache-2.0: https://www.apache.org/licenses/LICENSE-2.0

.. </legal notes>

methods and properties
=========================

*)

{attribute 'enable_dynamic_creation'}
FUNCTION_BLOCK ReverseOrderComparator EXTENDS CNM_ABstractObject.Object IMPLEMENTS CNM_AbstractObject.IComparator


(*

short summary
=================
This abstract property returns the class name of the concrete object, 
which is useful to check the class name for ``__DELETE``.

.. <legal notes>

legal notes
=================
| SPDX-FileCopyrightText: © 2022 ekvip automation GmbH <info@ekvip.de>
| SPDX-License-Identifier: Apache-2.0
| For details check: Apache-2.0_

.. _Apache-2.0: https://www.apache.org/licenses/LICENSE-2.0

.. </legal notes>

*)
PROPERTY className :CNM_AbstractObject.ClassName
GET
className := 'ReverseOrderComparator_Internal';
END_GET
END_PROPERTY


(*

short summary
=================
This method is used to create a new instance
of the object which has the same internal state as the object.
If the object is a container class, the references to the content objects
are not cloned for this there is the method `ICloneable.deepClone`.

If an object does not support cloning the return value is
``CNM_ReturnTypes.CloneResult.CLONE_IS_NOT_SUPPORTED``.

If there is not enough memory or the cloning fails because the
attribute enable dynamic creation was forgotten the return value is 
``CNM_ReturnTypes.CloneResult.FAILED``.

Only if the return value is ``CNM_ReturnTypes.CloneResult.SUCCESS``
the output ``clonedObject`` points to the new object
otherwise ``clonedObject`` is NULL.  

.. <legal notes>

legal notes
=================
| SPDX-FileCopyrightText: © 2024 ekvip automation GmbH <info@ekvip.de>
| SPDX-License-Identifier: Apache-2.0
| For details check: Apache-2.0_

.. _Apache-2.0: https://www.apache.org/licenses/LICENSE-2.0

.. </legal notes>

parameters
=================
:return:``CNM_ReturnTypes.CloneResult.SUCCESS``: new object clone was created,
	``CNM_ReturnTypes.CloneResult.FAILED``: object clone failed
	``CNM_ReturnTypes.CloneResult.CLONE_IS_NOT_SUPPORTED``: object does not support cloning

*)

METHOD clone	:CNM_AbstractObject.CNM_ReturnTypes.CloneResult
VAR_OUTPUT
	(* new object instance or NULL if somthing went wrong *)
	clonedObject	:CNM_AbstractObject.IObject;
END_VAR
VAR
	newComparator	:POINTER TO ReverseOrderComparator;
END_VAR
newComparator := __NEW(ReverseOrderComparator());

IF ((
		newComparator <> 0
	) AND_THEN (
		__QUERYINTERFACE(newComparator^,clonedObject)
	)
) THEN
	clone := CNM_ReturnTypes.CloneResult.SUCCESS;
ELSE
	clone := CNM_ReturnTypes.CloneResult.FAILED;
END_IF
END_METHOD


(*

short summary
=================
This method compares two objects, this is needed for sort orders.

.. <legal notes>

legal notes
=================
| SPDX-FileCopyrightText: © 2022 ekvip automation GmbH <info@ekvip.de>
| SPDX-License-Identifier: Apache-2.0
| For details check: Apache-2.0_

.. _Apache-2.0: https://www.apache.org/licenses/LICENSE-2.0

.. </legal notes>

parameters
=================
:return: ``SMALLER``: ``object1`` precedes in order,
	``EQUAL``: ``object1`` and ``object2`` at the same position in order,
	``GREATER``: ``object1`` is after in order. Checkout the library CNM_ReturnTypes.

*)
METHOD compare :CNM_AbstractObject.CNM_ReturnTypes.ComparationResult
VAR_INPUT
	(* first object to compare*)
	object1	:CNM_AbstractObject.IObject;
	(* second object to compare*)
	object2	:CNM_AbstractObject.IObject;
END_VAR
IF THIS^.isObjectValid(object1) THEN
	CASE object1.compareTo(object2) OF
		CNM_ReturnTypes.ComparationResult.GREATER:
			compare := CNM_ReturnTypes.ComparationResult.SMALLER;
		CNM_ReturnTypes.ComparationResult.SMALLER:
			compare := CNM_ReturnTypes.ComparationResult.GREATER;
		ELSE
			compare := CNM_ReturnTypes.ComparationResult.EQUAL;
	END_CASE
ELSIF THIS^.isObjectValid(object2) THEN
	CASE object2.compareTo(object1) OF
		CNM_ReturnTypes.ComparationResult.GREATER:
			compare := CNM_ReturnTypes.ComparationResult.GREATER;
		CNM_ReturnTypes.ComparationResult.SMALLER:
			compare := CNM_ReturnTypes.ComparationResult.SMALLER;
		ELSE
			compare := CNM_ReturnTypes.ComparationResult.EQUAL;
	END_CASE
ELSE 
	compare := CNM_ReturnTypes.ComparationResult.GREATER;
END_IF
END_METHOD

(*

short summary
=================
This method is used to create a new instance
of the object which has the same internal state as the object.
If the object is a container class, the references to the content objects
are cloned too.

If an object does not support cloning the return value is
``CNM_ReturnTypes.CloneResult.CLONE_IS_NOT_SUPPORTED``.

If there is not enough memory or the cloning fails because the
attribute enable dynamic creation was forgotten the return value is 
``CNM_ReturnTypes.CloneResult.FAILED``.
If something goes wrong, then this method must clean up everything
that has been cloned and free the memory again.
**The deepClone either works completely, or not at all**

Only if the return value is ``CNM_ReturnTypes.CloneResult.SUCCESS``
the output ``clonedObject`` points to the new object
otherwise ``clonedObject`` is NULL.  

.. attention:: 
	For derivations: **If a derived class needs ``deepClone`` this method must be overwritten.**
	and don't forget the attribute ``{attribute 'enable_dynamic_creation'}``, even for container content 

.. <legal notes>

legal notes
=================
| SPDX-FileCopyrightText: © 2024 ekvip automation GmbH <info@ekvip.de>
| SPDX-License-Identifier: Apache-2.0
| For details check: Apache-2.0_

.. _Apache-2.0: https://www.apache.org/licenses/LICENSE-2.0

.. </legal notes>

parameters
=================
:return:``CNM_ReturnTypes.CloneResult.SUCCESS``: new object clone was created,
``CNM_ReturnTypes.CloneResult.FAILED``: object clone failed
``CNM_ReturnTypes.CloneResult.CLONE_IS_NOT_SUPPORTED``: object does not support deep cloning

*)

METHOD deepClone :CNM_ReturnTypes.CloneResult
VAR_OUTPUT
	(* new object instance or NULL if somthing went wrong *)
	clonedObject	:CNM_AbstractObject.IObject;
END_VAR
deepClone := THIS^.clone(clonedObject => clonedObject);
END_METHOD

END_FUNCTION_BLOCK

// ---- AssertionTester/AssertionTests/ObjectAssertions/classes/ObjectAssertionsTests.TcPOU
(*
short summary
==================
This class tests all methods of Object assertions
with various combinations of inputs and checks expected 
outputs are satisfied or not

.. <legal notes>

legal notes
=================
| SPDX-FileCopyrightText: © 2022 ekvip automation GmbH <info@ekvip.de>
| SPDX-License-Identifier: Apache-2.0
| For details check: Apache-2.0_

.. _Apache-2.0: https://www.apache.org/licenses/LICENSE-2.0

.. </legal notes>

methods and properties
======================

*)


FUNCTION_BLOCK ObjectAssertionsTests EXTENDS AbstractAssertorTest
VAR

END_VAR
VAR CONSTANT
	(* prefix to unify the test names *)
	TEST_NAME_PREFIX				:STRING := 'assert.object.';
	(* NULL value for Assertions *)
	{attribute 'const_replaced'}
	{attribute 'displaymode':='hex'}
	NULL 							:__XWORD := 0;
	(* max value of a DWORD *)
	{attribute 'hide'}
	MAX_DWORD						:DWORD := 16#FFFF_FFFF;
	(* min value of a DWORD *)
	{attribute 'hide'}
	MIN_DWORD						:DWORD := 16#0000_0000;
	(* only the msb is set *)
	{attribute 'hide'}
	MSB_ONLY						:DWORD := 16#8000_0000;
	(* only the msb is set *)
	{attribute 'hide'}
	LSB_ONLY						:DWORD := 16#0000_0001;
	(* all bits set except the msb *)
	{attribute 'hide'}
	WITHOUT_MSB 					:DWORD := 16#7FFF_FFFF;
	(* for every nibble is the msb set only *)
	{attribute 'hide'}
	ALL_NIBBLE_MSB					:DWORD := 16#8888_8888;
	(* for every nibble is the msb unset only *)
	{attribute 'hide'}
	WITHOUT_NIBBLE_MSB				:DWORD := 16#7777_7777;
	(* for every nibble is the lsb set only *)
	{attribute 'hide'}
	ALL_NIBBLE_LSB					:DWORD := 16#1111_1111;
	(* every bit is set except the lsb *)
	{attribute 'hide'}
	LSB_IS_UNSET					:DWORD := 16#FFFF_FFFE;
	(* NULL value of DWordValue *)
	{warning disable C0228}
	DWORDVALUE_NULL 				:DWordValue(0);
	(* max vale of DWordValue *)
	DWORDVALUE_MAX					:DWordValue(MAX_DWORD);
	(* min vale of DWordValue *)
	DWORDVALUE_MIN					:DWordValue(MIN_DWORD);
	(* only the msb is set *)
	DWORDVALUE_MSB_ONLY				:DWordValue(MSB_ONLY);
	(* all bits set except the msb *)
	DWORDVALUE_WITHOUT_MSB 			:DWordValue(WITHOUT_MSB);
	(* for every nibble is the msb set only *)
	DWORDVALUE_ALL_NIBBLE_MSB		:DWordValue(ALL_NIBBLE_MSB);
	(* for every nibble is the msb unset only *)
	DWORDVALUE_WITHOUT_NIBBLE_MSB	:DWordValue(WITHOUT_NIBBLE_MSB);
	(* for every nibble is the lsb set only *)
	DWORDVALUE_ALL_NIBBLE_LSB		:DWordValue(ALL_NIBBLE_LSB);	
	(* every bit is set except the lsb *)
	DWORDVALUE_LSB_IS_UNSET			:DWordValue(LSB_IS_UNSET);
	(* only the msb is set *)
	DWORDVALUE_LSB_ONLY				:DWordValue(LSB_ONLY);
	{warning ensable C0228}
END_VAR

THIS^.runIsEqualTo();
THIS^.runIsNotEqualTo();
THIS^.runObjectIsValid();
THIS^.runObjectIsNull();
THIS^.runIsAfterInOrderTo();
THIS^.runIsEqualInOrderTo();
THIS^.runPrecedesInOrderTo();
THIS^.runSetComparator();

(*

short summary
==================
This test method is a helper function to create a unified test name

.. <legal notes>

legal notes
=================
| SPDX-FileCopyrightText: © 2022 ekvip automation GmbH <info@ekvip.de>
| SPDX-License-Identifier: Apache-2.0
| For details check: Apache-2.0_

.. _Apache-2.0: https://www.apache.org/licenses/LICENSE-2.0

.. </legal notes>

parameters
==========

*)

METHOD PROTECTED getTestNameFor :Tc2_System.T_MaxString
VAR_INPUT
	(* name of the method to test, to create a unified test name *)
	nameOfMethodToTest	:Tc2_System.T_MaxString;
END_VAR
getTestNameFor := Tc2_Standard.CONCAT(THIS^.TEST_NAME_PREFIX, nameOfMethodToTest);
END_METHOD

(*

short summary
==================
This test method tests ``assert.object.isAfterInOrderTo``
method of CNM_AssertionInterfaces library with various inputs

.. <legal notes>

legal notes
=================
| SPDX-FileCopyrightText: © 2022 ekvip automation GmbH <info@ekvip.de>
| SPDX-License-Identifier: Apache-2.0
| For details check: Apache-2.0_

.. _Apache-2.0: https://www.apache.org/licenses/LICENSE-2.0

.. </legal notes>

*)


METHOD runIsAfterInOrderTo
RETURN (NOT TcUnit.TEST_ORDERED(THIS^.getTestNameFor('isAfterInOrderTo')));

THIS^.testIsAfterInOrderTo(
	objectToTest := THIS^.DWORDVALUE_MAX,
	expectedObject := THIS^.DWORDVALUE_MAX
);
THIS^.testIsAfterInOrderTo(
	objectToTest := THIS^.DWORDVALUE_MIN,
	expectedObject := THIS^.DWORDVALUE_MIN
);
THIS^.testIsAfterInOrderTo(
	objectToTest := THIS^.DWORDVALUE_MIN,
	expectedObject := THIS^.DWORDVALUE_MAX
);
THIS^.testIsAfterInOrderTo(
	objectToTest := THIS^.DWORDVALUE_MAX,
	expectedObject := THIS^.DWORDVALUE_MIN
);
THIS^.testIsAfterInOrderTo(
	objectToTest := THIS^.DWORDVALUE_MAX,
	expectedObject := THIS^.DWORDVALUE_MIN
);
THIS^.testIsAfterInOrderTo(
	objectToTest := THIS^.DWORDVALUE_ALL_NIBBLE_LSB,
	expectedObject := THIS^.DWORDVALUE_ALL_NIBBLE_LSB
);
THIS^.testIsAfterInOrderTo(
	objectToTest := THIS^.DWORDVALUE_LSB_ONLY,
	expectedObject := THIS^.DWORDVALUE_MSB_ONLY
);
THIS^.testIsAfterInOrderTo(
	objectToTest := THIS^.DWORDVALUE_MSB_ONLY,
	expectedObject := THIS^.DWORDVALUE_MSB_ONLY
);
THIS^.testIsAfterInOrderTo(
	objectToTest := THIS^.DWORDVALUE_MSB_ONLY,
	expectedObject := THIS^.DWORDVALUE_LSB_ONLY
);
THIS^.testIsAfterInOrderTo(
	objectToTest := THIS^.DWORDVALUE_MIN,
	expectedObject := 0
);
THIS^.testIsAfterInOrderTo(
	objectToTest := 0,
	expectedObject := THIS^.DWORDVALUE_MAX
);

TcUnit.TEST_FINISHED();
END_METHOD

(*

short summary
==================
This test method tests ``assert.object.isEqualInOrderTo``
method of CNM_AssertionInterfaces library with various inputs

.. <legal notes>

legal notes
=================
| SPDX-FileCopyrightText: © 2022 ekvip automation GmbH <info@ekvip.de>
| SPDX-License-Identifier: Apache-2.0
| For details check: Apache-2.0_

.. _Apache-2.0: https://www.apache.org/licenses/LICENSE-2.0

.. </legal notes>

*)


METHOD runIsEqualInOrderTo
RETURN (NOT TcUnit.TEST_ORDERED(THIS^.getTestNameFor('isEqualInOrderTo')));

THIS^.testIsEqualInOrderTo(
	objectToTest := THIS^.DWORDVALUE_MAX,
	expectedObject := THIS^.DWORDVALUE_MAX
);
THIS^.testIsEqualInOrderTo(
	objectToTest := THIS^.DWORDVALUE_MIN,
	expectedObject := THIS^.DWORDVALUE_MIN
);
THIS^.testIsEqualInOrderTo(
	objectToTest := THIS^.DWORDVALUE_MIN,
	expectedObject := THIS^.DWORDVALUE_MAX
);
THIS^.testIsEqualInOrderTo(
	objectToTest := THIS^.DWORDVALUE_MAX,
	expectedObject := THIS^.DWORDVALUE_MIN
);
THIS^.testIsEqualInOrderTo(
	objectToTest := THIS^.DWORDVALUE_MAX,
	expectedObject := THIS^.DWORDVALUE_MIN
);
THIS^.testIsEqualInOrderTo(
	objectToTest := THIS^.DWORDVALUE_ALL_NIBBLE_LSB,
	expectedObject := THIS^.DWORDVALUE_ALL_NIBBLE_LSB
);
THIS^.testIsEqualInOrderTo(
	objectToTest := THIS^.DWORDVALUE_LSB_ONLY,
	expectedObject := THIS^.DWORDVALUE_MSB_ONLY
);
THIS^.testIsEqualInOrderTo(
	objectToTest := THIS^.DWORDVALUE_MSB_ONLY,
	expectedObject := THIS^.DWORDVALUE_MSB_ONLY
);
THIS^.testIsEqualInOrderTo(
	objectToTest := THIS^.DWORDVALUE_MSB_ONLY,
	expectedObject := THIS^.DWORDVALUE_LSB_ONLY
);
THIS^.testIsEqualInOrderTo(
	objectToTest := THIS^.DWORDVALUE_MIN,
	expectedObject := 0
);
THIS^.testIsEqualInOrderTo(
	objectToTest := 0,
	expectedObject := THIS^.DWORDVALUE_MAX
);

TcUnit.TEST_FINISHED();
END_METHOD

(*

short summary
==================
This test method tests ``assert.object.isEqualTo``
method of CNM_AssertionInterfaces library with various inputs

.. <legal notes>

legal notes
=================
| SPDX-FileCopyrightText: © 2022 ekvip automation GmbH <info@ekvip.de>
| SPDX-License-Identifier: Apache-2.0
| For details check: Apache-2.0_

.. _Apache-2.0: https://www.apache.org/licenses/LICENSE-2.0

.. </legal notes>

*)


METHOD runIsEqualTo
RETURN (NOT TcUnit.TEST_ORDERED(THIS^.getTestNameFor('isEqualTo')));

THIS^.testIsEqualTo(
	objectToTest := THIS^.DWORDVALUE_MAX,
	expectedObject := THIS^.DWORDVALUE_MAX
);
THIS^.testIsEqualTo(
	objectToTest := THIS^.DWORDVALUE_MIN,
	expectedObject := THIS^.DWORDVALUE_MIN
);
THIS^.testIsEqualTo(
	objectToTest := THIS^.DWORDVALUE_MIN,
	expectedObject := THIS^.DWORDVALUE_MAX
);
THIS^.testIsEqualTo(
	objectToTest := THIS^.DWORDVALUE_MAX,
	expectedObject := THIS^.DWORDVALUE_MIN
);
THIS^.testIsEqualTo(
	objectToTest := THIS^.DWORDVALUE_MAX,
	expectedObject := THIS^.DWORDVALUE_MIN
);
THIS^.testIsEqualTo(
	objectToTest := THIS^.DWORDVALUE_ALL_NIBBLE_LSB,
	expectedObject := THIS^.DWORDVALUE_ALL_NIBBLE_LSB
);
THIS^.testIsEqualTo(
	objectToTest := THIS^.DWORDVALUE_LSB_ONLY,
	expectedObject := THIS^.DWORDVALUE_MSB_ONLY
);
THIS^.testIsEqualTo(
	objectToTest := THIS^.DWORDVALUE_MSB_ONLY,
	expectedObject := THIS^.DWORDVALUE_MSB_ONLY
);
THIS^.testIsEqualTo(
	objectToTest := THIS^.DWORDVALUE_MSB_ONLY,
	expectedObject := THIS^.DWORDVALUE_LSB_ONLY
);
THIS^.testIsEqualTo(
	objectToTest := THIS^.DWORDVALUE_MIN,
	expectedObject := 0
);
THIS^.testIsEqualTo(
	objectToTest := 0,
	expectedObject := THIS^.DWORDVALUE_MAX
);

TcUnit.TEST_FINISHED();
END_METHOD

(*

short summary
==================
This test method tests ``assert.object.isNotEqualTo``
method of CNM_AssertionInterfaces library with various inputs

.. <legal notes>

legal notes
=================
| SPDX-FileCopyrightText: © 2022 ekvip automation GmbH <info@ekvip.de>
| SPDX-License-Identifier: Apache-2.0
| For details check: Apache-2.0_

.. _Apache-2.0: https://www.apache.org/licenses/LICENSE-2.0

.. </legal notes>

*)


METHOD runIsNotEqualTo
RETURN (NOT TcUnit.TEST_ORDERED(THIS^.getTestNameFor('isNotEqualTo')));

THIS^.testIsNotEqualTo(
	objectToTest := THIS^.DWORDVALUE_MAX,
	expectedObject := THIS^.DWORDVALUE_MAX
);
THIS^.testIsNotEqualTo(
	objectToTest := THIS^.DWORDVALUE_MIN,
	expectedObject := THIS^.DWORDVALUE_MIN
);
THIS^.testIsNotEqualTo(
	objectToTest := THIS^.DWORDVALUE_MIN,
	expectedObject := THIS^.DWORDVALUE_MAX
);
THIS^.testIsNotEqualTo(
	objectToTest := THIS^.DWORDVALUE_MAX,
	expectedObject := THIS^.DWORDVALUE_MIN
);
THIS^.testIsNotEqualTo(
	objectToTest := THIS^.DWORDVALUE_ALL_NIBBLE_LSB,
	expectedObject := THIS^.DWORDVALUE_ALL_NIBBLE_LSB
);
THIS^.testIsNotEqualTo(
	objectToTest := THIS^.DWORDVALUE_LSB_ONLY,
	expectedObject := THIS^.DWORDVALUE_MSB_ONLY
);
THIS^.testIsNotEqualTo(
	objectToTest := THIS^.DWORDVALUE_MSB_ONLY,
	expectedObject := THIS^.DWORDVALUE_MSB_ONLY
);
THIS^.testIsNotEqualTo(
	objectToTest := THIS^.DWORDVALUE_MSB_ONLY,
	expectedObject := THIS^.DWORDVALUE_LSB_ONLY
);
THIS^.testIsNotEqualTo(
	objectToTest := THIS^.DWORDVALUE_MIN,
	expectedObject := 0
);
THIS^.testIsNotEqualTo(
	objectToTest := 0,
	expectedObject := THIS^.DWORDVALUE_MAX
);

TcUnit.TEST_FINISHED();
END_METHOD

(*

short summary
==================
This test method tests ``assert.object.objectIsNull``
method of CNM_AssertionInterfaces library with various inputs

.. <legal notes>

legal notes
=================
| SPDX-FileCopyrightText: © 2022 ekvip automation GmbH <info@ekvip.de>
| SPDX-License-Identifier: Apache-2.0
| For details check: Apache-2.0_

.. _Apache-2.0: https://www.apache.org/licenses/LICENSE-2.0

.. </legal notes>

*)


METHOD runObjectIsNull
RETURN (NOT TcUnit.TEST_ORDERED(THIS^.getTestNameFor('objectIsNull')));

THIS^.testObjectIsNull(
	objectToTest := THIS^.DWORDVALUE_MAX
);
THIS^.testObjectIsNull(
	objectToTest := THIS^.DWORDVALUE_MIN
);
THIS^.testObjectIsNull(
	objectToTest := THIS^.DWORDVALUE_ALL_NIBBLE_LSB
);
THIS^.testObjectIsNull(
	objectToTest := THIS^.DWORDVALUE_LSB_ONLY
);
THIS^.testObjectIsNull(
	objectToTest := THIS^.DWORDVALUE_MSB_ONLY
);
THIS^.testObjectIsNull(
	objectToTest := 0
);

TcUnit.TEST_FINISHED();
END_METHOD

(*

short summary
==================
This test method tests ``assert.object.objectIsValid``
method of CNM_AssertionInterfaces library with various inputs

.. <legal notes>

legal notes
=================
| SPDX-FileCopyrightText: © 2022 ekvip automation GmbH <info@ekvip.de>
| SPDX-License-Identifier: Apache-2.0
| For details check: Apache-2.0_

.. _Apache-2.0: https://www.apache.org/licenses/LICENSE-2.0

.. </legal notes>

*)


METHOD runObjectIsValid
RETURN (NOT TcUnit.TEST_ORDERED(THIS^.getTestNameFor('objectIsValid')));

THIS^.testObjectIsValid(
	objectToTest := THIS^.DWORDVALUE_MAX
);
THIS^.testObjectIsValid(
	objectToTest := THIS^.DWORDVALUE_MIN
);
THIS^.testObjectIsValid(
	objectToTest := THIS^.DWORDVALUE_ALL_NIBBLE_LSB
);
THIS^.testObjectIsValid(
	objectToTest := THIS^.DWORDVALUE_LSB_ONLY
);
THIS^.testObjectIsValid(
	objectToTest := THIS^.DWORDVALUE_MSB_ONLY
);
THIS^.testObjectIsValid(
	objectToTest := 0
);

TcUnit.TEST_FINISHED();
END_METHOD

(*

short summary
==================
This test method tests ``assert.object.precedesInOrderTo``
method of CNM_AssertionInterfaces library with various inputs

.. <legal notes>

legal notes
=================
| SPDX-FileCopyrightText: © 2022 ekvip automation GmbH <info@ekvip.de>
| SPDX-License-Identifier: Apache-2.0
| For details check: Apache-2.0_

.. _Apache-2.0: https://www.apache.org/licenses/LICENSE-2.0

.. </legal notes>

*)


METHOD runPrecedesInOrderTo
RETURN (NOT TcUnit.TEST_ORDERED(THIS^.getTestNameFor('precedesInOrderTo')));

THIS^.testPrecedesInOrderTo(
	objectToTest := THIS^.DWORDVALUE_MAX,
	expectedObject := THIS^.DWORDVALUE_MAX
);
THIS^.testPrecedesInOrderTo(
	objectToTest := THIS^.DWORDVALUE_MIN,
	expectedObject := THIS^.DWORDVALUE_MIN
);
THIS^.testPrecedesInOrderTo(
	objectToTest := THIS^.DWORDVALUE_MIN,
	expectedObject := THIS^.DWORDVALUE_MAX
);
THIS^.testPrecedesInOrderTo(
	objectToTest := THIS^.DWORDVALUE_MAX,
	expectedObject := THIS^.DWORDVALUE_MIN
);
THIS^.testPrecedesInOrderTo(
	objectToTest := THIS^.DWORDVALUE_MAX,
	expectedObject := THIS^.DWORDVALUE_MIN
);
THIS^.testPrecedesInOrderTo(
	objectToTest := THIS^.DWORDVALUE_ALL_NIBBLE_LSB,
	expectedObject := THIS^.DWORDVALUE_ALL_NIBBLE_LSB
);
THIS^.testPrecedesInOrderTo(
	objectToTest := THIS^.DWORDVALUE_LSB_ONLY,
	expectedObject := THIS^.DWORDVALUE_MSB_ONLY
);
THIS^.testPrecedesInOrderTo(
	objectToTest := THIS^.DWORDVALUE_MSB_ONLY,
	expectedObject := THIS^.DWORDVALUE_MSB_ONLY
);
THIS^.testPrecedesInOrderTo(
	objectToTest := THIS^.DWORDVALUE_MSB_ONLY,
	expectedObject := THIS^.DWORDVALUE_LSB_ONLY
);
THIS^.testPrecedesInOrderTo(
	objectToTest := THIS^.DWORDVALUE_MIN,
	expectedObject := 0
);
THIS^.testPrecedesInOrderTo(
	objectToTest := 0,
	expectedObject := THIS^.DWORDVALUE_MAX
);

TcUnit.TEST_FINISHED();
END_METHOD

(*

short summary
==================
This test method tests ``assert.object.setComparator``
method of CNM_AssertionInterfaces library with various inputs

.. <legal notes>

legal notes
=================
| SPDX-FileCopyrightText: © 2022 ekvip automation GmbH <info@ekvip.de>
| SPDX-License-Identifier: Apache-2.0
| For details check: Apache-2.0_

.. _Apache-2.0: https://www.apache.org/licenses/LICENSE-2.0

.. </legal notes>

*)


METHOD runSetComparator
VAR
	reverseOrderComparator :ReverseOrderComparator;
END_VAR
RETURN (NOT TcUnit.TEST_ORDERED(THIS^.getTestNameFor('setComparator')));


THIS^.testSetComparator(
	objectToTest := THIS^.DWORDVALUE_MAX,
	expectedObject := THIS^.DWORDVALUE_MAX
);
THIS^.testSetComparator(
	objectToTest := THIS^.DWORDVALUE_MIN,
	expectedObject := THIS^.DWORDVALUE_MIN
);
THIS^.testSetComparator(
	objectToTest := THIS^.DWORDVALUE_MIN,
	expectedObject := THIS^.DWORDVALUE_MAX
);
THIS^.testSetComparator(
	objectToTest := THIS^.DWORDVALUE_MAX,
	expectedObject := THIS^.DWORDVALUE_MIN
);
THIS^.testSetComparator(
	objectToTest := THIS^.DWORDVALUE_MAX,
	expectedObject := THIS^.DWORDVALUE_MIN
);
THIS^.testSetComparator(
	objectToTest := THIS^.DWORDVALUE_ALL_NIBBLE_LSB,
	expectedObject := THIS^.DWORDVALUE_ALL_NIBBLE_LSB
);
THIS^.testSetComparator(
	objectToTest := THIS^.DWORDVALUE_LSB_ONLY,
	expectedObject := THIS^.DWORDVALUE_MSB_ONLY
);
THIS^.testSetComparator(
	objectToTest := THIS^.DWORDVALUE_MSB_ONLY,
	expectedObject := THIS^.DWORDVALUE_MSB_ONLY
);
THIS^.testSetComparator(
	objectToTest := THIS^.DWORDVALUE_MSB_ONLY,
	expectedObject := THIS^.DWORDVALUE_LSB_ONLY
);
THIS^.testSetComparator(
	objectToTest := THIS^.DWORDVALUE_MIN,
	expectedObject := 0
);
THIS^.testSetComparator(
	objectToTest := 0,
	expectedObject := THIS^.DWORDVALUE_MAX
);

TcUnit.TEST_FINISHED();
END_METHOD

(*

short summary
==================
This test method tests ``assert.object.isAfterInOrderTo``
method of CNM_AssertionInterfaces library, 
it provides the possibility to handover test data via parameter 


.. <legal notes>

legal notes
=================
| SPDX-FileCopyrightText: © 2022 ekvip automation GmbH <info@ekvip.de>
| SPDX-License-Identifier: Apache-2.0
| For details check: Apache-2.0_

.. _Apache-2.0: https://www.apache.org/licenses/LICENSE-2.0

.. </legal notes>

parameters
==========

*)


METHOD testIsAfterInOrderTo
VAR_INPUT
(* for the test it's the parameter ``object`` *)
	objectToTest	:IDWord;
	(* for the test it's the parameter ``objectToCompare`` *)
	expectedObject	:IDWord;
END_VAR
VAR
	(* just the expectation if the assertion to test must be worng or true *)
	assertionIsWrong		:BOOL;
	(* contains the format string for the test message *)
	message					:Tc2_System.T_MaxString;
	(* TwinCAT printf with the test message *)
	messageStringBuilder	:Tc2_Utilities.FB_FormatString;
	(* DWORD value of ``object`` as string *)
	objectToTestAsString	:STRING(22);
	(* DWORD value of ``objectToCompare`` as string *)
	expectedObjectAsString	:STRING(22);
	(* needed to call AbstractObject Methods on ´´DWordValue´´ *)
	concreteObject 			:ConcreteObject;
END_VAR
THIS^.assertorContainer.resetAssertor();

IF (
		concreteObject.isObjectValid(objectToTest)
) THEN
		assertionIsWrong := (objectToTest.compareTo(expectedObject) <> CNM_ReturnTypes.ComparationResult.GREATER);
ELSIF (
		concreteObject.isObjectValid(expectedObject)
) THEN
		assertionIsWrong := (expectedObject.compareTo(objectToTest) >= CNM_ReturnTypes.ComparationResult.EQUAL);
END_IF

message := SEL(
	assertionIsWrong,
	'object is %s objectToCompare is %s assertion must be TRUE', 
	'object is %s objectToCompare is %s assertion must be FALSE'
);

IF (
		concreteObject.isObjectValid(objectToTest)
) THEN
		objectToTestAsString := TO_STRING(objectToTest.value);
ELSE
		objectToTestAsString := 'NULL';
END_IF

IF (
		concreteObject.isObjectValid(expectedObject)
) THEN
		expectedObjectAsString := TO_STRING(expectedObject.value);
ELSE
		expectedObjectAsString := 'NULL';
END_IF

messageStringBuilder(
	sFormat := message,
	arg1 := THIS^.AnyToArg(objectToTestAsString),
	arg2 := THIS^.AnyToArg(expectedObjectAsString)
);


THIS^.assertorContainer.assertor.assert.object.isAfterInOrderTo(
	object	:= objectToTest,
	objectToCompare	:= expectedObject,
	message			:= ''
);

THIS^.AssertEquals_BOOL(
	Expected 	:= assertionIsWrong,
	Actual 		:= THIS^.assertorContainer.wasAssertionWrong,
	Message 	:= messageStringBuilder.sOut
);
END_METHOD

(*

short summary
==================
This test method tests ´´ReverseOrderComparator´´ in ``assert.object.setComparator``
method of CNM_AssertionInterfaces library, 
it provides the possibility to handover test data via parameter 


.. <legal notes>

legal notes
=================
| SPDX-FileCopyrightText: © 2022 ekvip automation GmbH <info@ekvip.de>
| SPDX-License-Identifier: Apache-2.0
| For details check: Apache-2.0_

.. _Apache-2.0: https://www.apache.org/licenses/LICENSE-2.0

.. </legal notes>

parameters
==========

*)


METHOD testIsAfterInOrderToReversed
VAR_INPUT
(* for the test it's the parameter ``object`` *)
	objectToTest	:IDWord;
	(* for the test it's the parameter ``objectToCompare`` *)
	expectedObject	:IDWord;
END_VAR
VAR
	(* just the expectation if the assertion to test must be worng or true *)
	assertionIsWrong		:BOOL;
	(* contains the format string for the test message *)
	message					:Tc2_System.T_MaxString;
	(* TwinCAT printf with the test message *)
	messageStringBuilder	:Tc2_Utilities.FB_FormatString;
	(* DWORD value of ``object`` as string *)
	objectToTestAsString	:STRING(22);
	(* DWORD value of ``objectToCompare`` as string *)
	expectedObjectAsString	:STRING(22);
	(* needed to call AbstractObject Methods on ´´DWordValue´´ *)
	concreteObject 			:ConcreteObject;
END_VAR
THIS^.assertorContainer.resetAssertor();

IF (
		concreteObject.isObjectValid(objectToTest)
) THEN
	assertionIsWrong := (objectToTest.compareTo(expectedObject) <> CNM_ReturnTypes.ComparationResult.SMALLER);
ELSIF (
		concreteObject.isObjectValid(expectedObject)
) THEN
	assertionIsWrong := (expectedObject.compareTo(objectToTest) <= CNM_ReturnTypes.ComparationResult.EQUAL);
END_IF

message := SEL(
	assertionIsWrong,
	'object is %s objectToCompare is %s assertion must be TRUE', 
	'object is %s objectToCompare is %s assertion must be FALSE'
);

IF (
		concreteObject.isObjectValid(objectToTest)
) THEN
	objectToTestAsString := TO_STRING(objectToTest.value);
ELSE
	objectToTestAsString := 'NULL';
END_IF

IF (
		concreteObject.isObjectValid(expectedObject)
) THEN
	expectedObjectAsString := TO_STRING(expectedObject.value);
ELSE
	expectedObjectAsString := 'NULL';
END_IF

messageStringBuilder(
	sFormat := message,
	arg1 := THIS^.AnyToArg(objectToTestAsString),
	arg2 := THIS^.AnyToArg(expectedObjectAsString)
);


THIS^.assertorContainer.assertor.assert.object.isAfterInOrderTo(
	object	:= objectToTest,
	objectToCompare	:= expectedObject,
	message			:= ''
);

THIS^.AssertEquals_BOOL(
	Expected 	:= assertionIsWrong,
	Actual 		:= THIS^.assertorContainer.wasAssertionWrong,
	Message 	:= messageStringBuilder.sOut
);
END_METHOD

(*

short summary
==================
This test method tests ``assert.object.isEqualInOrderTo``
method of CNM_AssertionInterfaces library, 
it provides the possibility to handover test data via parameter 


.. <legal notes>

legal notes
=================
| SPDX-FileCopyrightText: © 2022 ekvip automation GmbH <info@ekvip.de>
| SPDX-License-Identifier: Apache-2.0
| For details check: Apache-2.0_

.. _Apache-2.0: https://www.apache.org/licenses/LICENSE-2.0

.. </legal notes>

parameters
==========

*)


METHOD testIsEqualInOrderTo
VAR_INPUT
(* for the test it's the parameter ``object`` *)
	objectToTest	:IDWord;
	(* for the test it's the parameter ``objectToCompare`` *)
	expectedObject	:IDWord;
END_VAR
VAR
	(* just the expectation if the assertion to test must be worng or true *)
	assertionIsWrong		:BOOL;
	(* contains the format string for the test message *)
	message					:Tc2_System.T_MaxString;
	(* TwinCAT printf with the test message *)
	messageStringBuilder	:Tc2_Utilities.FB_FormatString;
	(* DWORD value of ``object`` as string *)
	objectToTestAsString	:STRING(22);
	(* DWORD value of ``objectToCompare`` as string *)
	expectedObjectAsString	:STRING(22);
	(* needed to call AbstractObject Methods on ´´DWordValue´´ *)
	concreteObject 			:ConcreteObject;
END_VAR
THIS^.assertorContainer.resetAssertor();

IF (
		concreteObject.isObjectValid(objectToTest)
) THEN
	assertionIsWrong := (objectToTest.compareTo(expectedObject) <> CNM_ReturnTypes.ComparationResult.EQUAL);
ELSIF (
		concreteObject.isObjectValid(expectedObject)
) THEN
	assertionIsWrong := (expectedObject.compareTo(objectToTest) <> CNM_ReturnTypes.ComparationResult.EQUAL);
END_IF

message := SEL(
	assertionIsWrong,
	'object is %s objectToCompare is %s assertion must be TRUE', 
	'object is %s objectToCompare is %s assertion must be FALSE'
);

IF (
		concreteObject.isObjectValid(objectToTest)
) THEN
	objectToTestAsString := TO_STRING(objectToTest.value);
ELSE
	objectToTestAsString := 'NULL';
END_IF

IF (
		concreteObject.isObjectValid(expectedObject)
) THEN
	expectedObjectAsString := TO_STRING(expectedObject.value);
ELSE
	expectedObjectAsString := 'NULL';
END_IF

messageStringBuilder(
	sFormat := message,
	arg1 := THIS^.AnyToArg(objectToTestAsString),
	arg2 := THIS^.AnyToArg(expectedObjectAsString)
);


THIS^.assertorContainer.assertor.assert.object.isEqualInOrderTo(
	object	:= objectToTest,
	objectToCompare	:= expectedObject,
	message			:= ''
);

THIS^.AssertEquals_BOOL(
	Expected 	:= assertionIsWrong,
	Actual 		:= THIS^.assertorContainer.wasAssertionWrong,
	Message 	:= messageStringBuilder.sOut
);
END_METHOD

(*

short summary
==================
This test method tests ´´ReverseOrderComparator´´ in ``assert.object.setComparator``
method of CNM_AssertionInterfaces library, 
it provides the possibility to handover test data via parameter 


.. <legal notes>

legal notes
=================
| SPDX-FileCopyrightText: © 2022 ekvip automation GmbH <info@ekvip.de>
| SPDX-License-Identifier: Apache-2.0
| For details check: Apache-2.0_

.. _Apache-2.0: https://www.apache.org/licenses/LICENSE-2.0

.. </legal notes>

parameters
==========

*)


METHOD testIsEqualInOrderToReversed
VAR_INPUT
(* for the test it's the parameter ``object`` *)
	objectToTest	:IDWord;
	(* for the test it's the parameter ``objectToCompare`` *)
	expectedObject	:IDWord;
END_VAR
VAR
	(* just the expectation if the assertion to test must be worng or true *)
	assertionIsWrong		:BOOL;
	(* contains the format string for the test message *)
	message					:Tc2_System.T_MaxString;
	(* TwinCAT printf with the test message *)
	messageStringBuilder	:Tc2_Utilities.FB_FormatString;
	(* DWORD value of ``object`` as string *)
	objectToTestAsString	:STRING(22);
	(* DWORD value of ``objectToCompare`` as string *)
	expectedObjectAsString	:STRING(22);
	(* needed to call AbstractObject Methods on ´´DWordValue´´ *)
	concreteObject 			:ConcreteObject;
END_VAR
THIS^.assertorContainer.resetAssertor();

IF (
		concreteObject.isObjectValid(objectToTest)
) THEN
	assertionIsWrong := (objectToTest.compareTo(expectedObject) <> CNM_ReturnTypes.ComparationResult.EQUAL);
ELSIF (
		concreteObject.isObjectValid(expectedObject)
) THEN
	assertionIsWrong := (expectedObject.compareTo(objectToTest) <> CNM_ReturnTypes.ComparationResult.EQUAL);
END_IF

message := SEL(
	assertionIsWrong,
	'object is %s objectToCompare is %s assertion must be TRUE', 
	'object is %s objectToCompare is %s assertion must be FALSE'
);

IF (
		concreteObject.isObjectValid(objectToTest)
) THEN
	objectToTestAsString := TO_STRING(objectToTest.value);
ELSE
	objectToTestAsString := 'NULL';
END_IF

IF (
		concreteObject.isObjectValid(expectedObject)
) THEN
	expectedObjectAsString := TO_STRING(expectedObject.value);
ELSE
	expectedObjectAsString := 'NULL';
END_IF

messageStringBuilder(
	sFormat := message,
	arg1 := THIS^.AnyToArg(objectToTestAsString),
	arg2 := THIS^.AnyToArg(expectedObjectAsString)
);


THIS^.assertorContainer.assertor.assert.object.isEqualInOrderTo(
	object	:= objectToTest,
	objectToCompare	:= expectedObject,
	message			:= ''
);

THIS^.AssertEquals_BOOL(
	Expected 	:= assertionIsWrong,
	Actual 		:= THIS^.assertorContainer.wasAssertionWrong,
	Message 	:= messageStringBuilder.sOut
);
END_METHOD

(*

short summary
==================
This test method tests ``assert.object.isEqualTo``
method of CNM_AssertionInterfaces library, 
it provides the possibility to handover test data via parameter 


.. <legal notes>

legal notes
=================
| SPDX-FileCopyrightText: © 2022 ekvip automation GmbH <info@ekvip.de>
| SPDX-License-Identifier: Apache-2.0
| For details check: Apache-2.0_

.. _Apache-2.0: https://www.apache.org/licenses/LICENSE-2.0

.. </legal notes>

parameters
==========

*)


METHOD testIsEqualTo
VAR_INPUT
(* for the test it's the parameter ``object`` *)
	objectToTest	:IDWord;
	(* for the test it's the parameter ``objectToCompare`` *)
	expectedObject	:IDWord;
END_VAR
VAR
	(* just the expectation if the assertion to test must be worng or true *)
	assertionIsWrong		:BOOL;
	(* contains the format string for the test message *)
	message					:Tc2_System.T_MaxString;
	(* TwinCAT printf with the test message *)
	messageStringBuilder	:Tc2_Utilities.FB_FormatString;
	(* DWORD value of ``object`` as string *)
	objectToTestAsString	:STRING(22);
	(* DWORD value of ``objectToCompare`` as string *)
	expectedObjectAsString	:STRING(22);
	(* needed to call AbstractObject Methods on ´´DWordValue´´ *)
	concreteObject 			:ConcreteObject;
END_VAR
THIS^.assertorContainer.resetAssertor();

IF (
		concreteObject.isObjectValid(objectToTest)
) THEN
	assertionIsWrong := (NOT objectToTest.isEqual(expectedObject));
ELSIF (
		concreteObject.isObjectValid(expectedObject)
) THEN
	assertionIsWrong := (NOT expectedObject.isEqual(objectToTest));
END_IF

message := SEL(
	assertionIsWrong,
	'object is %s objectToCompare is %s assertion must be TRUE', 
	'object is %s objectToCompare is %s assertion must be FALSE'
);

IF (
		concreteObject.isObjectValid(objectToTest)
) THEN
	objectToTestAsString := TO_STRING(objectToTest.value);
ELSE
	objectToTestAsString := 'NULL';
END_IF

IF (
		concreteObject.isObjectValid(expectedObject)
) THEN
	expectedObjectAsString := TO_STRING(expectedObject.value);
ELSE
	expectedObjectAsString := 'NULL';
END_IF

messageStringBuilder(
	sFormat := message,
	arg1 := THIS^.AnyToArg(objectToTestAsString),
	arg2 := THIS^.AnyToArg(expectedObjectAsString)
);


THIS^.assertorContainer.assertor.assert.object.isEqualTo(
	object	:= objectToTest,
	objectToCompare	:= expectedObject,
	message			:= ''
);

THIS^.AssertEquals_BOOL(
	Expected 	:= assertionIsWrong,
	Actual 		:= THIS^.assertorContainer.wasAssertionWrong,
	Message 	:= messageStringBuilder.sOut
);
END_METHOD

(*

short summary
==================
This test method tests ``assert.object.isNotEqualTo``
method of CNM_AssertionInterfaces library, 
it provides the possibility to handover test data via parameter 


.. <legal notes>

legal notes
=================
| SPDX-FileCopyrightText: © 2022 ekvip automation GmbH <info@ekvip.de>
| SPDX-License-Identifier: Apache-2.0
| For details check: Apache-2.0_

.. _Apache-2.0: https://www.apache.org/licenses/LICENSE-2.0

.. </legal notes>

parameters
==========

*)


METHOD testIsNotEqualTo
VAR_INPUT
(* for the test it's the parameter ``object`` *)
	objectToTest	:IDWord;
	(* for the test it's the parameter ``objectToCompare`` *)
	expectedObject	:IDWord;
END_VAR
VAR
	(* just the expectation if the assertion to test must be worng or true *)
	assertionIsWrong		:BOOL;
	(* contains the format string for the test message *)
	message					:Tc2_System.T_MaxString;
	(* TwinCAT printf with the test message *)
	messageStringBuilder	:Tc2_Utilities.FB_FormatString;
	(* DWORD value of ``object`` as string *)
	objectToTestAsString	:STRING(22);
	(* DWORD value of ``objectToCompare`` as string *)
	expectedObjectAsString	:STRING(22);
	(* needed to call AbstractObject Methods on ´´DWordValue´´ *)
	concreteObject 			:ConcreteObject;
END_VAR
THIS^.assertorContainer.resetAssertor();

IF (
		concreteObject.isObjectValid(objectToTest)
) THEN
	assertionIsWrong := (objectToTest.isEqual(expectedObject));
ELSIF (concreteObject.isObjectValid(expectedObject)) THEN
		assertionIsWrong := (expectedObject.isEqual(objectToTest));
END_IF

message := SEL(
	assertionIsWrong,
	'object is %s objectToCompare is %s assertion must be TRUE', 
	'object is %s objectToCompare is %s assertion must be FALSE'
);

IF (
		concreteObject.isObjectValid(objectToTest)
) THEN
	objectToTestAsString := TO_STRING(objectToTest.value);
ELSE
	objectToTestAsString := 'NULL';
END_IF

IF (
		concreteObject.isObjectValid(expectedObject)
) THEN
	expectedObjectAsString := TO_STRING(expectedObject.value);
ELSE
	expectedObjectAsString := 'NULL';
END_IF

messageStringBuilder(
	sFormat := message,
	arg1 := THIS^.AnyToArg(objectToTestAsString),
	arg2 := THIS^.AnyToArg(expectedObjectAsString)
);


THIS^.assertorContainer.assertor.assert.object.isNotEqualTo(
	object	:= objectToTest,
	objectToCompare	:= expectedObject,
	message			:= ''
);

THIS^.AssertEquals_BOOL(
	Expected 	:= assertionIsWrong,
	Actual 		:= THIS^.assertorContainer.wasAssertionWrong,
	Message 	:= messageStringBuilder.sOut
);
END_METHOD

(*

short summary
==================
This test method tests ``assert.object.objectIsNull``
method of CNM_AssertionInterfaces library, 
it provides the possibility to handover test data via parameter 


.. <legal notes>

legal notes
=================
| SPDX-FileCopyrightText: © 2022 ekvip automation GmbH <info@ekvip.de>
| SPDX-License-Identifier: Apache-2.0
| For details check: Apache-2.0_

.. _Apache-2.0: https://www.apache.org/licenses/LICENSE-2.0

.. </legal notes>

parameters
==========

*)


METHOD testObjectIsNull
VAR_INPUT
(* for the test it's the parameter ``object`` *)
	objectToTest	:IDWord;
END_VAR
VAR
	(* just the expectation if the assertion to test must be worng or true *)
	assertionIsWrong		:BOOL;
	(* contains the format string for the test message *)
	message					:Tc2_System.T_MaxString;
	(* TwinCAT printf with the test message *)
	messageStringBuilder	:Tc2_Utilities.FB_FormatString;
	(* DWORD value of ``object`` as string *)
	objectToTestAsString	:STRING(22);
	(* needed to call AbstractObject Methods on ´´DWordValue´´ *)
	concreteObject 			:ConcreteObject;
END_VAR
THIS^.assertorContainer.resetAssertor();

assertionIsWrong := (concreteObject.isObjectValid(objectToTest));

message := SEL(
	assertionIsWrong,
	'object is %s expected is NOT NULL assertion must be TRUE', 
	'object is %s expected is NULL assertion must be FALSE'
);

IF (
		concreteObject.isObjectValid(objectToTest)
) THEN
	objectToTestAsString := TO_STRING(objectToTest.value);
ELSE
	objectToTestAsString := 'NULL';
END_IF

messageStringBuilder(
	sFormat := message,
	arg1 := THIS^.AnyToArg(objectToTestAsString),
);

THIS^.assertorContainer.assertor.assert.object.objectIsNull(
	object	:= objectToTest,
	message			:= ''
);

THIS^.AssertEquals_BOOL(
	Expected 	:= assertionIsWrong,
	Actual 		:= THIS^.assertorContainer.wasAssertionWrong,
	Message 	:= messageStringBuilder.sOut
);
END_METHOD

(*

short summary
==================
This test method tests ``assert.object.objectIsValid``
method of CNM_AssertionInterfaces library, 
it provides the possibility to handover test data via parameter 


.. <legal notes>

legal notes
=================
| SPDX-FileCopyrightText: © 2022 ekvip automation GmbH <info@ekvip.de>
| SPDX-License-Identifier: Apache-2.0
| For details check: Apache-2.0_

.. _Apache-2.0: https://www.apache.org/licenses/LICENSE-2.0

.. </legal notes>

parameters
==========

*)


METHOD testObjectIsValid
VAR_INPUT
(* for the test it's the parameter ``object`` *)
	objectToTest	:IDWord;
END_VAR
VAR
	(* just the expectation if the assertion to test must be worng or true *)
	assertionIsWrong		:BOOL;
	(* contains the format string for the test message *)
	message					:Tc2_System.T_MaxString;
	(* TwinCAT printf with the test message *)
	messageStringBuilder	:Tc2_Utilities.FB_FormatString;
	(* DWORD value of ``object`` as string *)
	objectToTestAsString	:STRING(22);
	(* needed to call AbstractObject Methods on ´´DWordValue´´ *)
	concreteObject 			:ConcreteObject;
END_VAR
THIS^.assertorContainer.resetAssertor();

assertionIsWrong := (NOT concreteObject.isObjectValid(objectToTest));

message := SEL(
	assertionIsWrong,
	'object is %s expected is NULL assertion must be TRUE', 
	'object is %s expected is NOT NULL assertion must be FALSE'
);

IF (
		concreteObject.isObjectValid(objectToTest)
) THEN
	objectToTestAsString := TO_STRING(objectToTest.value);
ELSE
	objectToTestAsString := 'NULL';
END_IF

messageStringBuilder(
	sFormat := message,
	arg1 := THIS^.AnyToArg(objectToTestAsString),
);

THIS^.assertorContainer.assertor.assert.object.objectIsValid(
	object	:= objectToTest,
	message			:= ''
);

THIS^.AssertEquals_BOOL(
	Expected 	:= assertionIsWrong,
	Actual 		:= THIS^.assertorContainer.wasAssertionWrong,
	Message 	:= messageStringBuilder.sOut
);
END_METHOD

(*

short summary
==================
This test method tests ``assert.object.precedesInOrderTo``
method of CNM_AssertionInterfaces library, 
it provides the possibility to handover test data via parameter 


.. <legal notes>

legal notes
=================
| SPDX-FileCopyrightText: © 2022 ekvip automation GmbH <info@ekvip.de>
| SPDX-License-Identifier: Apache-2.0
| For details check: Apache-2.0_

.. _Apache-2.0: https://www.apache.org/licenses/LICENSE-2.0

.. </legal notes>

parameters
==========

*)


METHOD testPrecedesInOrderTo
VAR_INPUT
(* for the test it's the parameter ``object`` *)
	objectToTest	:IDWord;
	(* for the test it's the parameter ``objectToCompare`` *)
	expectedObject	:IDWord;
END_VAR
VAR
	(* just the expectation if the assertion to test must be worng or true *)
	assertionIsWrong		:BOOL;
	(* contains the format string for the test message *)
	message					:Tc2_System.T_MaxString;
	(* TwinCAT printf with the test message *)
	messageStringBuilder	:Tc2_Utilities.FB_FormatString;
	(* DWORD value of ``object`` as string *)
	objectToTestAsString	:STRING(22);
	(* DWORD value of ``objectToCompare`` as string *)
	expectedObjectAsString	:STRING(22);
	(* needed to call AbstractObject Methods on ´´DWordValue´´ *)
	concreteObject 			:ConcreteObject;
END_VAR
THIS^.assertorContainer.resetAssertor();

IF (
		concreteObject.isObjectValid(objectToTest)
) THEN
	assertionIsWrong := (objectToTest.compareTo(expectedObject) <> CNM_ReturnTypes.ComparationResult.SMALLER);
ELSIF (
		concreteObject.isObjectValid(expectedObject)
) THEN
	assertionIsWrong := (expectedObject.compareTo(objectToTest) <= CNM_ReturnTypes.ComparationResult.EQUAL);
END_IF

message := SEL(
	assertionIsWrong,
	'object is %s objectToCompare is %s assertion must be TRUE', 
	'object is %s objectToCompare is %s assertion must be FALSE'
);

IF (
		concreteObject.isObjectValid(objectToTest)
) THEN
	objectToTestAsString := TO_STRING(objectToTest.value);
ELSE
	objectToTestAsString := 'NULL';
END_IF

IF (
		concreteObject.isObjectValid(expectedObject)
) THEN
	expectedObjectAsString := TO_STRING(expectedObject.value);
ELSE
	expectedObjectAsString := 'NULL';
END_IF

messageStringBuilder(
	sFormat := message,
	arg1 := THIS^.AnyToArg(objectToTestAsString),
	arg2 := THIS^.AnyToArg(expectedObjectAsString)
);


THIS^.assertorContainer.assertor.assert.object.precedesInOrderTo(
	object	:= objectToTest,
	objectToCompare	:= expectedObject,
	message			:= ''
);

THIS^.AssertEquals_BOOL(
	Expected 	:= assertionIsWrong,
	Actual 		:= THIS^.assertorContainer.wasAssertionWrong,
	Message 	:= messageStringBuilder.sOut
);
END_METHOD

(*

short summary
==================
This test method tests ´´ReverseOrderComparator´´ in ``assert.object.setComparator``
method of CNM_AssertionInterfaces library, 
it provides the possibility to handover test data via parameter 


.. <legal notes>

legal notes
=================
| SPDX-FileCopyrightText: © 2022 ekvip automation GmbH <info@ekvip.de>
| SPDX-License-Identifier: Apache-2.0
| For details check: Apache-2.0_

.. _Apache-2.0: https://www.apache.org/licenses/LICENSE-2.0

.. </legal notes>

parameters
==========

*)


METHOD testPrecedesInOrderToReversed
VAR_INPUT
(* for the test it's the parameter ``object`` *)
	objectToTest	:IDWord;
	(* for the test it's the parameter ``objectToCompare`` *)
	expectedObject	:IDWord;
END_VAR
VAR
	(* just the expectation if the assertion to test must be worng or true *)
	assertionIsWrong		:BOOL;
	(* contains the format string for the test message *)
	message					:Tc2_System.T_MaxString;
	(* TwinCAT printf with the test message *)
	messageStringBuilder	:Tc2_Utilities.FB_FormatString;
	(* DWORD value of ``object`` as string *)
	objectToTestAsString	:STRING(22);
	(* DWORD value of ``objectToCompare`` as string *)
	expectedObjectAsString	:STRING(22);
	(* needed to call AbstractObject Methods on ´´DWordValue´´ *)
	concreteObject 			:ConcreteObject;
END_VAR
THIS^.assertorContainer.resetAssertor();

IF (
		concreteObject.isObjectValid(objectToTest)
) THEN
	assertionIsWrong := (objectToTest.compareTo(expectedObject) <> CNM_ReturnTypes.ComparationResult.GREATER);
ELSIF (
		concreteObject.isObjectValid(expectedObject)
) THEN
	assertionIsWrong := (expectedObject.compareTo(objectToTest) >= CNM_ReturnTypes.ComparationResult.EQUAL);
END_IF

message := SEL(
	assertionIsWrong,
	'object is %s objectToCompare is %s assertion must be TRUE', 
	'object is %s objectToCompare is %s assertion must be FALSE'
);

IF (
		concreteObject.isObjectValid(objectToTest)
) THEN
	objectToTestAsString := TO_STRING(objectToTest.value);
ELSE
	objectToTestAsString := 'NULL';
END_IF

IF (
		concreteObject.isObjectValid(expectedObject)
) THEN
	expectedObjectAsString := TO_STRING(expectedObject.value);
ELSE
	expectedObjectAsString := 'NULL';
END_IF

messageStringBuilder(
	sFormat := message,
	arg1 := THIS^.AnyToArg(objectToTestAsString),
	arg2 := THIS^.AnyToArg(expectedObjectAsString)
);


THIS^.assertorContainer.assertor.assert.object.precedesInOrderTo(
	object	:= objectToTest,
	objectToCompare	:= expectedObject,
	message			:= ''
);

THIS^.AssertEquals_BOOL(
	Expected 	:= assertionIsWrong,
	Actual 		:= THIS^.assertorContainer.wasAssertionWrong,
	Message 	:= messageStringBuilder.sOut
);
END_METHOD

(*

short summary
==================
This test method tests ``assert.object.setComparator``
method of CNM_AssertionInterfaces library, 
it provides the possibility to handover test data via parameter 


.. <legal notes>

legal notes
=================
| SPDX-FileCopyrightText: © 2022 ekvip automation GmbH <info@ekvip.de>
| SPDX-License-Identifier: Apache-2.0
| For details check: Apache-2.0_

.. _Apache-2.0: https://www.apache.org/licenses/LICENSE-2.0

.. </legal notes>

parameters
==========

*)


METHOD testSetComparator
VAR_INPUT
(* for the test it's the parameter ``object`` *)
	objectToTest	:IDWord;
	(* for the test it's the parameter ``objectToCompare`` *)
	expectedObject	:IDWord;
END_VAR
VAR
	(* just the expectation if the assertion to test must be worng or true *)
	assertionIsWrong		:BOOL;
	(* contains the format string for the test message *)
	message					:Tc2_System.T_MaxString;
	(* TwinCAT printf with the test message *)
	messageStringBuilder	:Tc2_Utilities.FB_FormatString;
	(* DWORD value of ``object`` as string *)
	objectToTestAsString	:STRING(22);
	(* DWORD value of ``objectToCompare`` as string *)
	expectedObjectAsString	:STRING(22);
	(* needed to call AbstractObject Methods on ´´DWordValue´´ *)
	concreteObject 			:ConcreteObject;
	(* this comparaotr will be set: compares in reversed order *)
	reverseOrderComparator 	:ReverseOrderComparator;
END_VAR
THIS^.assertorContainer.resetAssertor();

//	set ReverseOrderComparator as comparator
THIS^.assertorContainer.assertor.assert.object.setComperator(
	comperator := reverseOrderComparator
);

//	test if comparator was set to ReverseOrderComparator
THIS^.testPrecedesInOrderToReversed(
	objectToTest := objectToTest,
	expectedObject := expectedObject
);
THIS^.testIsEqualInOrderToReversed(
	objectToTest := objectToTest,
	expectedObject := expectedObject
);
THIS^.testIsAfterInOrderToReversed(
	objectToTest := objectToTest,
	expectedObject := expectedObject
);

//	unset ReverseOrderComparator
THIS^.assertorContainer.assertor.assert.object.setComperator(
	comperator := 0
);

// test if comparator was reseted
THIS^.testPrecedesInOrderTo(
	objectToTest := objectToTest,
	expectedObject := expectedObject
);
THIS^.testIsEqualInOrderTo(
	objectToTest := objectToTest,
	expectedObject := expectedObject
);
THIS^.testIsAfterInOrderTo(
	objectToTest := objectToTest,
	expectedObject := expectedObject
);
END_METHOD

END_FUNCTION_BLOCK

// ---- AssertionTester/AssertionTests/PointerAssertions/classes/PointerAssertionsTests.TcPOU
(*

short summary
=================
This class designed for the Unit Tests of Assertions Class Library. Each method is testing the Assertion Class's methods with different input and expect different outputs.
The message of the test output is extended version of method itself.

.. <legal notes>

legal notes
=================
| SPDX-FileCopyrightText: © 2022 ekvip automation GmbH <info@ekvip.de>
| SPDX-License-Identifier: Apache-2.0
| For details check: Apache-2.0_

.. _Apache-2.0: https://www.apache.org/licenses/LICENSE-2.0

.. </legal notes>

methods and properties
=======================

*)

FUNCTION_BLOCK PointerAssertionsTests EXTENDS AbstractAssertorTest
VAR
	(* pointer to dynamic allocated memory with one byte *)
	oneByte							:POINTER TO BYTE;
	(* pointer to a dynmic allocated array with the size of ``ARRAY_SIZE`` *)
	byteArray						:POINTER TO BYTE;
	(* cnc function block to create cnc data *)
	{attribute 'hide'}
	hli								:Tc2_CncHli.MCV_HliInterface;
	(* pointer to a cnc memory area *)
	cncAddress						:POINTER TO Tc2_CncHli.HLI_V_E_DATA;
	(* size of cnc object *)
	cncSize							:UDINT;
	(* alternative this pointer *)
	me								:POINTER TO PointerAssertionsTests := THIS;
	(* weired THIS pointer *)
	itsMeAgain						:POINTER TO POINTER TO PointerAssertionsTests := ADR(me);
	(* alternative Super pointer *)
	myMom							:POINTER TO AbstractAssertorTest := SUPER;
	(* invalid pointer to dynamic allocated memory *)
	invalidByte						:POINTER TO BYTE;
END_VAR
VAR CONSTANT
	(* prefix to unify the test names *)
	TEST_NAME_PREFIX		:Tc2_System.T_MaxString := 'assert.pointers.';
	(* contains no address	*)
	NULL_POINTER			:PVOID := 0;
	(* size of this test class *)
	I_AM_FAT				:UDINT := SIZEOF(PointerAssertionsTests);
	(* just zero to test with valid pointer but size zero *)
	SIZE_ZERO				:UDINT := 0;
	(* size of dynamic byte array *)
	ARRAY_SIZE				:UDINT := 15;
	(* since we don't know the lenght of a POINTER we need it to initialize ``INVALID_POINTER`` *)
	{attribute 'hide'}
	INIT_INVALID_POINTER	:__XWORD := 16#FFFF_FFFF;
	(* just a non null invalid ``POINTER`` *)
	INVALID_POINTER			:PVOID := 16#20;//(ROR(INIT_INVALID_POINTER, 32) OR INIT_INVALID_POINTER);
	(* 0x400000 is 4096kb and this is the max configurable stack size *)
	{attribute 'displaymode':='hex'}
	MAX_STACK_SIZE :__XWORD := 16#0040_0000;
END_VAR

THIS^.init();
THIS^.runIsAlignedTests();
THIS^.runIsDwordAlignedTests();
THIS^.runIsLwordAlignedTests();
THIS^.runIsNotNullTests();
THIS^.runIsNullTests();
THIS^.runIsNotOverlappingTests();
THIS^.runIsOverlappingTests();
THIS^.runIsEqualToTests();
THIS^.runIsNotEqualToTests();
THIS^.runIsValidTests();
THIS^.runMemoryAreaIsCncTests();
THIS^.runMemoryAreaIsDynamicTests();
THIS^.runMemoryAreaIsStaticTests();
THIS^.runMemoryAreaIsUnknownTests();
THIS^.runMemoryAreaIsNotCncTests();
THIS^.runMemoryAreaIsNotDynamicTests();
THIS^.runMemoryAreaIsNotStaticTests();
THIS^.runMemoryAreaIsNotUnknownTests();
THIS^.leave();

(*

short summary
=============

.. <legal notes>

legal notes
=================
| SPDX-FileCopyrightText: © 2023 ekvip automation GmbH <info@ekvip.de>
| SPDX-License-Identifier: Apache-2.0
| For details check: Apache-2.0_

.. _Apache-2.0: https://www.apache.org/licenses/LICENSE-2.0

.. </legal notes>

parameters
==========

*)

METHOD FB_exit : BOOL
VAR_INPUT
	bInCopyCode : BOOL; // if TRUE, the exit method is called for exiting an instance that is copied afterwards (online change).
END_VAR
THIS^.leave();
END_METHOD

METHOD FB_reinit : BOOL
VAR_INPUT
END_VAR
THIS^.leave();
THIS^.init();
END_METHOD

(*

short summary
==================
This test method is a helper function to create a unified test name

.. <legal notes>

legal notes
=================
| SPDX-FileCopyrightText: © 2022 ekvip automation GmbH <info@ekvip.de>
| SPDX-License-Identifier: Apache-2.0
| For details check: Apache-2.0_

.. _Apache-2.0: https://www.apache.org/licenses/LICENSE-2.0

.. </legal notes>

parameters
==========

*)

METHOD PROTECTED getTestNameFor :Tc2_System.T_MaxString
VAR_INPUT
	(* name of the method to test, to create a unified test name *)
	nameOfMethodToTest	:Tc2_System.T_MaxString;
END_VAR
getTestNameFor := Tc2_Standard.CONCAT(THIS^.TEST_NAME_PREFIX, nameOfMethodToTest);
END_METHOD

(*

short summary
==================
it initilaze dynamic and cnc pointers

.. <legal notes>

legal notes
=================
| SPDX-FileCopyrightText: © 2022 ekvip automation GmbH <info@ekvip.de>
| SPDX-License-Identifier: Apache-2.0
| For details check: Apache-2.0_

.. _Apache-2.0: https://www.apache.org/licenses/LICENSE-2.0

.. </legal notes>

parameters
==========

*)

METHOD PROTECTED init
VAR_INPUT
END_VAR
VAR
	(* this is just a dummy pointer to create an invalid dynamic pointer *)
	dmy	:POINTER TO BYTE;
END_VAR
THIS^.hli();
THIS^.cncAddress := Tc2_CncHli.HLI_Global_Variables.gpVEGlobal;
THIS^.cncSize := Tc2_CncHli.HLI_Global_Variables.gVEGlobMemSize;
THIS^.oneByte := __NEW(BYTE);
THIS^.byteArray := __NEW(BYTE, THIS^.ARRAY_SIZE);
dmy := __NEW(BYTE);
THIS^.invalidByte := dmy;
__DELETE(dmy);
END_METHOD

(*

short summary
==================
it free the memory of dynamic pointers again

.. <legal notes>

legal notes
=================
| SPDX-FileCopyrightText: © 2022 ekvip automation GmbH <info@ekvip.de>
| SPDX-License-Identifier: Apache-2.0
| For details check: Apache-2.0_

.. _Apache-2.0: https://www.apache.org/licenses/LICENSE-2.0

.. </legal notes>

parameters
==========

*)

METHOD PROTECTED leave
VAR_INPUT
END_VAR
IF (THIS^.oneByte <> 0) THEN
	__DELETE(THIS^.oneByte);
END_IF
IF (THIS^.byteArray <> 0) THEN
	__DELETE(THIS^.byteArray);
END_IF
END_METHOD

METHOD PROTECTED memoryAreaToString :Tc2_System.T_MaxString
VAR_INPUT
	area	:Tc2_System.E_TcMemoryArea;
END_VAR
CASE area OF
Tc2_System.E_TcMemoryArea.CNC: memoryAreaToString := 'CNC';
Tc2_System.E_TcMemoryArea.Dynamic: memoryAreaToString := 'Dynamic';
Tc2_System.E_TcMemoryArea.Static: memoryAreaToString := 'Static';
ELSE memoryAreaToString := 'Unkown';
END_CASE
END_METHOD

(*

short summary
==================
This test method tests ``assert.pointers.isAligned``
method of CNM_AssertionInterfaces library with various inputs

.. <legal notes>

legal notes
=================
| SPDX-FileCopyrightText: © 2022 ekvip automation GmbH <info@ekvip.de>
| SPDX-License-Identifier: Apache-2.0
| For details check: Apache-2.0_

.. _Apache-2.0: https://www.apache.org/licenses/LICENSE-2.0

.. _Apache-2.THIS^.SIZE_ZERO: https://www.apache.org/licenses/LICENSE-2.THIS^.SIZE_ZERO

.. </legal notes>

*)

METHOD runIsAlignedTests
VAR
	foo				:XWORD;
	stackAddress	:PVOID;
END_VAR
RETURN (NOT TcUnit.TEST_ORDERED(THIS^.getTestNameFor('isAligned')));
stackAddress := ADR(foo);

THIS^.testIsAligned(
	address := THIS,
);
THIS^.testIsAligned(
	address := THIS^.NULL_POINTER,
);
THIS^.testIsAligned(
	address := THIS^.NULL_POINTER + 1,
);
THIS^.testIsAligned(
	address := stackAddress,
);
THIS^.testIsAligned(
	address := stackAddress + 3,
);
THIS^.testIsAligned(
	address := THIS^.oneByte,
);
THIS^.testIsAligned(
	address := THIS^.oneByte + 7,
);
THIS^.testIsAligned(
	address := THIS^.byteArray,
);
THIS^.testIsAligned(
	address := THIS^.byteArray + 2,
);
THIS^.testIsAligned(
	address := THIS^.cncAddress,
);
THIS^.testIsAligned(
	address := THIS^.cncAddress + 1,
);
THIS^.testIsAligned(
	address := THIS^.itsMeAgain,
);
THIS^.testIsAligned(
	address := THIS^.itsMeAgain + 6,
);
THIS^.testIsAligned(
	address := THIS^.me,
);
THIS^.testIsAligned(
	address := THIS^.me + 3,
);
THIS^.testIsAligned(
	address := THIS^.myMom,
);
THIS^.testIsAligned(
	address := THIS^.invalidByte,
);
THIS^.testIsAligned(
	address := THIS^.invalidByte + 4,
);
THIS^.testIsAligned(
	address := THIS^.INVALID_POINTER,
);
THIS^.testIsAligned(
	address := THIS^.INVALID_POINTER + 1,
);

TcUnit.TEST_FINISHED();
END_METHOD

(*

short summary
==================
This test method tests ``assert.pointers.isDwordAligned``
method of CNM_AssertionInterfaces library with various inputs

.. <legal notes>

